C03638=1065.158,313.293,401.347,173.947,33.225,156.127
C03639=1065.152,313.045,401.379,173.944,33.220,156.126
C03640=1065.146,312.797,401.412,173.941,33.216,156.125
C03641=1065.139,312.550,401.445,173.938,33.212,156.124
C03642=1065.133,312.302,401.478,173.934,33.207,156.124
C03643=1065.126,312.054,401.509,173.931,33.203,156.123
C03644=1065.120,311.806,401.542,173.928,33.199,156.122
C03645=1065.113,311.558,401.575,173.925,33.195,156.121
C03646=1065.107,311.311,401.608,173.922,33.190,156.120
C03647=1065.101,311.063,401.640,173.919,33.186,156.119
C03648=1065.094,310.816,401.673,173.915,33.181,156.118
C03649=1065.088,310.568,401.706,173.912,33.177,156.118
C03650=1065.082,310.320,401.738,173.909,33.173,156.117
C03651=1065.076,310.072,401.771,173.906,33.169,156.116
C03652=1065.069,309.824,401.804,173.903,33.165,156.115
C03653=1065.062,309.577,401.836,173.900,33.160,156.114
C03654=1065.056,309.328,401.868,173.897,33.156,156.113
C03655=1065.050,309.081,401.901,173.894,33.151,156.113
C03656=1065.043,308.833,401.933,173.890,33.147,156.112
C03657=1065.037,308.585,401.966,173.887,33.143,156.111
C03658=1065.031,308.337,401.998,173.884,33.139,156.110
C03659=1065.025,308.090,402.031,173.881,33.134,156.109
C03660=1065.019,307.842,402.063,173.877,33.130,156.108
C03661=1065.012,307.594,402.095,173.874,33.126,156.108
C03662=1065.005,307.347,402.128,173.871,33.121,156.107
C03663=1064.999,307.099,402.160,173.868,33.117,156.106
C03664=1064.993,306.851,402.193,173.865,33.113,156.105
C03665=1064.987,306.603,402.225,173.862,33.109,156.104
C03666=1064.981,306.355,402.257,173.859,33.104,156.103
C03667=1064.974,306.108,402.290,173.855,33.100,156.103
C03668=1064.968,305.860,402.322,173.852,33.095,156.102
C03669=1064.962,305.613,402.354,173.849,33.091,156.101
C03670=1064.956,305.365,402.386,173.846,33.087,156.100
C03671=1064.950,305.117,402.419,173.843,33.083,156.099
C03672=1064.943,304.882,402.449,173.840,33.079,156.099
C03673=1064.938,304.648,402.479,173.837,33.074,156.098
C03674=1064.932,304.413,402.510,173.835,33.071,156.097
C03675=1064.927,304.179,402.540,173.832,33.067,156.096
C03676=1064.920,303.944,402.571,173.829,33.062,156.095
C03677=1064.914,303.710,402.600,173.826,33.058,156.095
C03678=1064.908,303.476,402.631,173.823,33.055,156.094
C03679=1064.903,303.241,402.661,173.820,33.050,156.093
C03680=1064.897,302.994,402.694,173.817,33.046,156.092
C03681=1064.890,302.746,402.726,173.814,33.042,156.091
C03682=1064.884,302.498,402.758,173.811,33.038,156.091
C03683=1064.878,302.250,402.790,173.808,33.033,156.090
C03684=1064.872,302.002,402.822,173.805,33.029,156.089
C03685=1064.866,301.755,402.853,173.802,33.025,156.088
C03686=1064.860,301.506,402.885,173.799,33.021,156.087
C03687=1064.853,301.259,402.918,173.796,33.016,156.086
C03688=1064.847,301.011,402.950,173.793,33.012,156.086
C03689=1064.841,300.763,402.981,173.790,33.008,156.085
C03690=1064.835,300.515,403.013,173.787,33.003,156.084
C03691=1064.829,300.268,403.046,173.784,32.999,156.083
C03692=1064.824,300.020,403.078,173.781,32.995,156.082
C03693=1064.817,299.772,403.109,173.778,32.991,156.082
C03694=1064.811,299.524,403.141,173.775,32.986,156.081
C03695=1064.805,299.276,403.173,173.772,32.982,156.080
C03696=1064.800,299.028,403.205,173.769,32.978,156.079
C03697=1064.793,298.780,403.236,173.766,32.974,156.078
C03698=1064.787,298.532,403.268,173.763,32.970,156.077
C03699=1064.781,298.285,403.300,173.760,32.965,156.077
C03700=1064.775,298.037,403.331,173.757,32.961,156.076
C03701=1064.769,297.788,403.363,173.754,32.957,156.075
C03702=1064.763,297.541,403.395,173.751,32.953,156.074
C03703=1064.756,297.294,403.427,173.748,32.948,156.073
C03704=1064.751,297.045,403.459,173.745,32.944,156.073
C03705=1064.745,296.798,403.490,173.742,32.940,156.072
C03706=1064.739,296.549,403.522,173.739,32.936,156.071
C03707=1064.732,296.301,403.553,173.737,32.932,156.070
C03708=1064.726,296.053,403.585,173.734,32.927,156.069
C03709=1064.720,295.806,403.616,173.731,32.923,156.069
C03710=1064.714,295.558,403.648,173.728,32.919,156.068
C03711=1064.707,295.310,403.680,173.725,32.915,156.067
C03712=1064.702,295.062,403.711,173.722,32.911,156.066
C03713=1064.695,294.814,403.742,173.719,32.907,156.065
C03714=1064.688,294.566,403.773,173.716,32.902,156.065
C03715=1064.683,294.319,403.805,173.713,32.898,156.064
C03716=1064.676,294.071,403.837,173.710,32.894,156.063
C03717=1064.670,293.822,403.867,173.707,32.890,156.062
C03718=1064.664,293.575,403.898,173.704,32.886,156.061
C03719=1064.658,293.327,403.930,173.701,32.882,156.061
C03720=1064.651,293.078,403.961,173.698,32.878,156.060
C03721=1064.645,292.831,403.992,173.695,32.873,156.059
C03722=1064.639,292.583,404.024,173.692,32.870,156.058
C03723=1064.633,292.335,404.055,173.690,32.865,156.058
C03724=1064.625,292.001,404.096,173.686,32.860,156.056
C03725=1064.617,291.668,404.139,173.682,32.855,156.055
C03726=1064.609,291.334,404.181,173.678,32.848,156.054
C03727=1064.600,291.000,404.223,173.674,32.843,156.053
C03728=1064.591,290.631,404.269,173.670,32.837,156.052
C03729=1064.582,290.264,404.316,173.665,32.831,156.051
C03730=1064.572,289.896,404.361,173.661,32.825,156.050
C03731=1064.563,289.528,404.407,173.657,32.819,156.049
C03732=1064.557,289.280,404.438,173.654,32.815,156.048
C03733=1064.551,289.032,404.468,173.651,32.811,156.047
C03734=1064.545,288.784,404.500,173.648,32.807,156.046
C03735=1064.539,288.536,404.531,173.645,32.802,156.046
C03736=1064.532,288.288,404.562,173.642,32.799,156.045
C03737=1064.527,288.040,404.593,173.639,32.794,156.044
C03738=1064.520,287.792,404.623,173.637,32.790,156.043
C03739=1064.514,287.545,404.654,173.634,32.786,156.043
C03740=1064.508,287.296,404.685,173.631,32.782,156.042
C03741=1064.502,287.048,404.715,173.628,32.778,156.041
C03742=1064.495,286.800,404.747,173.625,32.774,156.040
C03743=1064.489,286.553,404.777,173.622,32.770,156.039
C03744=1064.483,286.304,404.808,173.620,32.766,156.039
C03745=1064.477,286.056,404.838,173.618,32.762,156.038
C03746=1064.470,285.808,404.870,173.615,32.758,156.037
C03747=1064.464,285.560,404.900,173.612,32.754,156.036
C03748=1064.458,285.312,404.931,173.609,32.750,156.036
C03749=1064.452,285.064,404.961,173.606,32.746,156.035
C03750=1064.446,284.816,404.992,173.603,32.742,156.034
C03751=1064.440,284.568,405.023,173.601,32.738,156.033
C03752=1064.434,284.321,405.053,173.598,32.734,156.033
C03753=1064.427,284.072,405.084,173.595,32.730,156.032
C03754=1064.422,283.824,405.114,173.592,32.726,156.031
C03755=1064.415,283.576,405.145,173.589,32.722,156.030
C03756=1064.409,283.328,405.175,173.586,32.718,156.030
C03757=1064.404,283.080,405.206,173.584,32.713,156.029
C03758=1064.397,282.832,405.236,173.581,32.710,156.028
C03759=1064.391,282.584,405.267,173.578,32.705,156.027
C03760=1064.385,282.335,405.298,173.575,32.701,156.026
C03761=1064.379,282.087,405.328,173.572,32.697,156.026
C03762=1064.373,281.840,405.358,173.570,32.693,156.025
C03763=1064.366,281.591,405.388,173.567,32.689,156.024
C03764=1064.360,281.344,405.419,173.564,32.685,156.023
C03765=1064.355,281.096,405.449,173.561,32.681,156.023
C03766=1064.348,280.847,405.480,173.558,32.677,156.022
C03767=1064.342,280.599,405.510,173.556,32.673,156.021
C03768=1064.336,280.352,405.540,173.553,32.669,156.020
C03769=1064.330,280.103,405.571,173.550,32.665,156.020
C03770=1064.324,279.855,405.602,173.547,32.661,156.019
C03771=1064.318,279.608,405.631,173.545,32.657,156.018
C03772=1064.311,279.359,405.662,173.543,32.653,156.017
C03773=1064.306,279.111,405.692,173.540,32.649,156.017
C03774=1064.300,278.863,405.722,173.537,32.645,156.016
C03775=1064.293,278.615,405.752,173.534,32.641,156.015
C03776=1064.287,278.367,405.782,173.532,32.637,156.014
C03777=1064.281,278.119,405.813,173.529,32.633,156.014
C03778=1064.274,277.870,405.842,173.526,32.629,156.013
C03779=1064.268,277.622,405.873,173.523,32.625,156.012
C03780=1064.263,277.401,405.900,173.521,32.621,156.011
C03781=1064.257,277.179,405.927,173.518,32.618,156.011
C03782=1064.252,276.958,405.953,173.516,32.614,156.010
C03783=1064.247,276.736,405.980,173.514,32.611,156.009
C03784=1064.242,276.514,406.007,173.511,32.607,156.009
C03785=1064.236,276.293,406.034,173.509,32.603,156.008
C03786=1064.230,276.071,406.060,173.506,32.600,156.007
C03787=1064.224,275.850,406.088,173.504,32.597,156.007
C03788=1064.219,275.601,406.117,173.501,32.592,156.006
C03789=1064.213,275.353,406.148,173.498,32.589,156.005
C03790=1064.207,275.105,406.177,173.496,32.585,156.005
C03791=1064.200,274.857,406.207,173.493,32.581,156.004
C03792=1064.194,274.609,406.237,173.490,32.577,156.003
C03793=1064.188,274.361,406.267,173.488,32.573,156.002
C03794=1064.182,274.113,406.297,173.486,32.569,156.002
C03795=1064.176,273.865,406.326,173.483,32.565,156.001
C03796=1064.170,273.616,406.357,173.480,32.561,156.000
C03797=1064.164,273.368,406.386,173.477,32.556,155.999
C03798=1064.158,273.120,406.416,173.475,32.553,155.999
C03799=1064.152,272.872,406.446,173.472,32.548,155.998
C03800=1064.146,272.624,406.476,173.469,32.545,155.997
C03801=1064.140,272.375,406.506,173.467,32.541,155.996
C03802=1064.133,272.128,406.535,173.464,32.537,155.996
C03803=1064.127,271.880,406.564,173.461,32.533,155.995
C03804=1064.121,271.631,406.594,173.459,32.529,155.994
C03805=1064.115,271.384,406.624,173.456,32.525,155.993
C03806=1064.109,271.135,406.653,173.453,32.521,155.993
C03807=1064.102,270.886,406.683,173.450,32.517,155.992
C03808=1064.097,270.639,406.713,173.448,32.513,155.991
C03809=1064.090,270.390,406.742,173.445,32.509,155.991
C03810=1064.085,270.142,406.772,173.443,32.505,155.990
C03811=1064.078,269.894,406.802,173.441,32.501,155.989
C03812=1064.072,269.646,406.831,173.438,32.497,155.988
C03813=1064.066,269.398,406.860,173.435,32.493,155.988
C03814=1064.060,269.150,406.889,173.433,32.490,155.987
C03815=1064.054,268.901,406.920,173.430,32.485,155.986
C03816=1064.048,268.653,406.949,173.427,32.481,155.985
C03817=1064.041,268.405,406.978,173.425,32.477,155.985
C03818=1064.036,268.157,407.008,173.422,32.474,155.984
C03819=1064.030,267.908,407.037,173.419,32.469,155.983
C03820=1064.023,267.661,407.067,173.417,32.466,155.982
C03821=1064.017,267.412,407.096,173.414,32.462,155.982
C03822=1064.011,267.164,407.125,173.411,32.458,155.981
C03823=1064.005,266.916,407.154,173.409,32.454,155.980
C03824=1063.999,266.668,407.183,173.406,32.450,155.979
C03825=1063.993,266.420,407.213,173.404,32.446,155.979
C03826=1063.987,266.171,407.242,173.402,32.442,155.978
C03827=1063.980,265.923,407.271,173.399,32.438,155.977
C03828=1063.975,265.674,407.301,173.396,32.434,155.977
C03829=1063.968,265.426,407.330,173.394,32.430,155.976
C03830=1063.962,265.178,407.359,173.391,32.426,155.975
C03831=1063.956,264.930,407.388,173.389,32.422,155.974
C03832=1063.950,264.681,407.418,173.386,32.418,155.974
C03833=1063.944,264.433,407.447,173.383,32.414,155.973
C03834=1063.938,264.185,407.476,173.381,32.410,155.972
C03835=1063.932,263.937,407.505,173.378,32.406,155.971
C03836=1063.926,263.718,407.531,173.376,32.403,155.971
C03837=1063.921,263.498,407.557,173.373,32.399,155.970
C03838=1063.916,263.278,407.583,173.371,32.396,155.969
C03839=1063.910,263.058,407.608,173.370,32.393,155.969
C03840=1063.905,262.838,407.634,173.367,32.389,155.968
C03841=1063.899,262.619,407.659,173.365,32.386,155.968
C03842=1063.894,262.398,407.685,173.363,32.382,155.967
C03843=1063.888,262.179,407.710,173.360,32.379,155.966
C03844=1063.882,261.930,407.739,173.358,32.375,155.966
C03845=1063.875,261.682,407.768,173.355,32.371,155.965
C03846=1063.869,261.434,407.797,173.353,32.367,155.964
C03847=1063.863,261.185,407.826,173.350,32.364,155.964
C03848=1063.857,260.937,407.855,173.347,32.359,155.963
C03849=1063.851,260.689,407.884,173.345,32.356,155.962
C03850=1063.844,260.441,407.913,173.342,32.352,155.961
C03851=1063.838,260.192,407.941,173.340,32.348,155.961
C03852=1063.832,259.944,407.970,173.338,32.344,155.960
C03853=1063.826,259.696,407.999,173.335,32.340,155.959
C03854=1063.819,259.448,408.028,173.333,32.336,155.958
C03855=1063.813,259.199,408.056,173.330,32.332,155.958
C03856=1063.807,258.951,408.085,173.328,32.328,155.957
C03857=1063.801,258.703,408.113,173.325,32.324,155.956
C03858=1063.795,258.455,408.142,173.322,32.320,155.956
C03859=1063.789,258.207,408.171,173.320,32.317,155.955
C03860=1063.783,257.958,408.199,173.317,32.313,155.954
C03861=1063.777,257.710,408.228,173.315,32.309,155.953
C03862=1063.771,257.461,408.257,173.312,32.305,155.953
C03863=1063.764,257.214,408.285,173.310,32.301,155.952
C03864=1063.758,256.965,408.314,173.308,32.297,155.951
C03865=1063.752,256.717,408.343,173.305,32.293,155.951
C03866=1063.745,256.469,408.372,173.303,32.289,155.950
C03867=1063.740,256.221,408.400,173.300,32.285,155.949
C03868=1063.734,255.972,408.429,173.298,32.282,155.948
C03869=1063.728,255.724,408.457,173.295,32.277,155.948
C03870=1063.721,255.476,408.485,173.293,32.274,155.947
C03871=1063.715,255.227,408.514,173.290,32.270,155.946
C03872=1063.709,254.979,408.543,173.288,32.266,155.946
C03873=1063.703,254.730,408.571,173.285,32.262,155.945
C03874=1063.697,254.482,408.599,173.283,32.258,155.944
C03875=1063.691,254.234,408.628,173.281,32.254,155.943
C03876=1063.685,253.985,408.656,173.278,32.250,155.943
C03877=1063.678,253.737,408.685,173.276,32.246,155.942
C03878=1063.672,253.489,408.713,173.273,32.242,155.941
C03879=1063.667,253.241,408.741,173.271,32.238,155.941
C03880=1063.661,252.992,408.770,173.268,32.234,155.940
C03881=1063.655,252.744,408.798,173.266,32.231,155.939
C03882=1063.648,252.495,408.826,173.263,32.226,155.938
C03883=1063.642,252.248,408.855,173.261,32.223,155.938
C03884=1063.636,251.999,408.883,173.259,32.219,155.937
C03885=1063.630,251.750,408.911,173.257,32.215,155.936
C03886=1063.625,251.502,408.940,173.254,32.211,155.935
C03887=1063.619,251.254,408.968,173.252,32.207,155.935
C03888=1063.612,251.006,408.996,173.249,32.203,155.934
C03889=1063.606,250.757,409.025,173.247,32.199,155.933
C03890=1063.601,250.509,409.053,173.244,32.195,155.933
C03891=1063.595,250.261,409.082,173.242,32.191,155.932
C03892=1063.589,250.040,409.106,173.240,32.187,155.931
C03893=1063.584,249.819,409.131,173.237,32.184,155.931
C03894=1063.578,249.598,409.157,173.236,32.181,155.930
C03895=1063.574,249.378,409.182,173.234,32.177,155.929
C03896=1063.568,249.157,409.207,173.232,32.173,155.929
C03897=1063.563,248.935,409.231,173.230,32.170,155.928
C03898=1063.558,248.714,409.256,173.227,32.166,155.927
C03899=1063.552,248.493,409.282,173.225,32.163,155.927
C03900=1063.546,248.245,409.309,173.223,32.158,155.926
C03901=1063.540,247.997,409.338,173.220,32.155,155.925
C03902=1063.534,247.748,409.367,173.218,32.150,155.924
C03903=1063.529,247.500,409.394,173.215,32.147,155.924
C03904=1063.522,247.252,409.422,173.214,32.142,155.923
C03905=1063.517,247.004,409.450,173.211,32.139,155.922
C03906=1063.511,246.755,409.478,173.209,32.135,155.922
C03907=1063.505,246.506,409.507,173.206,32.131,155.921
C03908=1063.499,246.259,409.534,173.204,32.127,155.920
C03909=1063.493,246.010,409.562,173.202,32.123,155.919
C03910=1063.486,245.761,409.590,173.199,32.119,155.919
C03911=1063.481,245.513,409.618,173.197,32.115,155.918
C03912=1063.474,245.265,409.646,173.194,32.111,155.917
C03913=1063.469,245.017,409.674,173.193,32.107,155.916
C03914=1063.462,244.768,409.701,173.190,32.103,155.916
C03915=1063.456,244.519,409.729,173.188,32.099,155.915
C03916=1063.450,244.271,409.757,173.185,32.095,155.914
C03917=1063.444,244.023,409.785,173.183,32.091,155.914
C03918=1063.438,243.775,409.812,173.181,32.088,155.913
C03919=1063.432,243.526,409.841,173.178,32.083,155.912
C03920=1063.426,243.278,409.868,173.176,32.080,155.911
C03921=1063.421,243.029,409.896,173.174,32.076,155.911
C03922=1063.414,242.781,409.923,173.172,32.072,155.910
C03923=1063.409,242.532,409.951,173.169,32.068,155.909
C03924=1063.402,242.284,409.979,173.167,32.063,155.908
C03925=1063.397,242.036,410.007,173.165,32.060,155.908
C03926=1063.390,241.787,410.034,173.162,32.056,155.907
C03927=1063.384,241.538,410.062,173.160,32.052,155.906
C03928=1063.378,241.290,410.090,173.157,32.048,155.906
C03929=1063.372,241.041,410.117,173.155,32.044,155.905
C03930=1063.366,240.794,410.144,173.154,32.040,155.904
C03931=1063.359,240.545,410.172,173.151,32.036,155.904
C03932=1063.354,240.297,410.199,173.149,32.033,155.903
C03933=1063.347,240.048,410.227,173.146,32.028,155.902
C03934=1063.341,239.800,410.254,173.144,32.025,155.901
C03935=1063.336,239.551,410.282,173.141,32.021,155.901
C03936=1063.329,239.303,410.309,173.139,32.017,155.900
C03937=1063.323,239.054,410.336,173.137,32.013,155.899
C03938=1063.317,238.806,410.364,173.135,32.008,155.898
C03939=1063.311,238.558,410.392,173.133,32.005,155.898
C03940=1063.305,238.309,410.419,173.131,32.001,155.897
C03941=1063.299,238.061,410.446,173.128,31.997,155.896
C03942=1063.292,237.812,410.473,173.126,31.993,155.896
C03943=1063.286,237.564,410.501,173.123,31.989,155.895
C03944=1063.281,237.315,410.528,173.121,31.985,155.894
C03945=1063.275,237.067,410.555,173.120,31.981,155.893
C03946=1063.268,236.818,410.583,173.117,31.978,155.893
C03947=1063.262,236.570,410.610,173.115,31.973,155.892
C03948=1063.257,236.345,410.634,173.113,31.970,155.891
C03949=1063.251,236.121,410.659,173.111,31.966,155.891
C03950=1063.246,235.898,410.684,173.108,31.963,155.890
C03951=1063.241,235.673,410.708,173.106,31.959,155.889
C03952=1063.235,235.449,410.733,173.104,31.955,155.889
C03953=1063.230,235.226,410.757,173.103,31.952,155.888
C03954=1063.224,235.002,410.781,173.101,31.949,155.888
C03955=1063.219,234.777,410.806,173.099,31.945,155.887
C03956=1063.213,234.529,410.833,173.096,31.940,155.886
C03957=1063.206,234.281,410.861,173.094,31.937,155.885
C03958=1063.201,234.032,410.887,173.092,31.933,155.885
C03959=1063.195,233.784,410.914,173.089,31.929,155.884
C03960=1063.189,233.535,410.942,173.087,31.925,155.883
C03961=1063.183,233.287,410.969,173.086,31.921,155.882
C03962=1063.177,233.038,410.996,173.083,31.917,155.882
C03963=1063.171,232.790,411.023,173.081,31.913,155.881
C03964=1063.165,232.542,411.050,173.079,31.909,155.880
C03965=1063.159,232.293,411.077,173.076,31.905,155.880
C03966=1063.153,232.044,411.104,173.074,31.901,155.879
C03967=1063.147,231.796,411.131,173.072,31.897,155.878
C03968=1063.140,231.547,411.158,173.070,31.893,155.877
C03969=1063.135,231.299,411.185,173.068,31.889,155.877
C03970=1063.129,231.051,411.211,173.066,31.886,155.876
C03971=1063.122,230.802,411.238,173.063,31.881,155.875
C03972=1063.116,230.554,411.266,173.061,31.877,155.875
C03973=1063.111,230.305,411.292,173.059,31.873,155.874
C03974=1063.104,230.056,411.319,173.056,31.869,155.873
C03975=1063.098,229.808,411.346,173.055,31.865,155.872
C03976=1063.093,229.560,411.373,173.053,31.861,155.872
C03977=1063.086,229.311,411.400,173.051,31.858,155.871
C03978=1063.080,229.062,411.426,173.048,31.853,155.870
C03979=1063.074,228.813,411.453,173.046,31.850,155.870
C03980=1063.068,228.565,411.480,173.044,31.845,155.869
C03981=1063.062,228.317,411.506,173.042,31.842,155.868
C03982=1063.055,228.068,411.533,173.040,31.838,155.867
C03983=1063.050,227.819,411.560,173.038,31.834,155.867
C03984=1063.044,227.571,411.586,173.035,31.830,155.866
C03985=1063.038,227.322,411.613,173.033,31.826,155.865
C03986=1063.031,227.074,411.640,173.031,31.822,155.864
C03987=1063.025,226.826,411.666,173.029,31.818,155.864
C03988=1063.019,226.577,411.693,173.027,31.814,155.863
C03989=1063.013,226.328,411.720,173.025,31.810,155.862
C03990=1063.007,226.080,411.747,173.023,31.806,155.862
C03991=1063.001,225.832,411.773,173.020,31.802,155.861
C03992=1062.994,225.583,411.800,173.018,31.798,155.860
C03993=1062.989,225.334,411.826,173.016,31.794,155.859
C03994=1062.983,225.086,411.853,173.014,31.790,155.859
C03995=1062.976,224.838,411.879,173.012,31.786,155.858
C03996=1062.970,224.589,411.906,173.010,31.782,155.857
C03997=1062.964,224.340,411.933,173.008,31.778,155.857
C03998=1062.959,224.091,411.959,173.005,31.774,155.856
C03999=1062.953,223.843,411.985,173.003,31.770,155.855
C04000=1062.946,223.595,412.011,173.001,31.766,155.854
C04001=1062.940,223.346,412.038,173.000,31.762,155.854
C04002=1062.934,223.098,412.065,172.997,31.758,155.853
C04003=1062.929,222.849,412.091,172.995,31.754,155.852
C04004=1062.923,222.621,412.115,172.993,31.751,155.852
C04005=1062.917,222.393,412.139,172.991,31.747,155.851
C04006=1062.913,222.165,412.163,172.989,31.743,155.850
C04007=1062.906,221.937,412.188,172.988,31.740,155.850
C04008=1062.901,221.709,412.212,172.986,31.736,155.849
C04009=1062.896,221.481,412.236,172.984,31.732,155.848
C04010=1062.890,221.253,412.260,172.982,31.728,155.848
C04011=1062.884,221.025,412.285,172.980,31.725,155.847
C04012=1062.878,220.777,412.311,172.978,31.720,155.846
C04013=1062.872,220.528,412.337,172.976,31.717,155.845
C04014=1062.866,220.279,412.363,172.974,31.713,155.845
C04015=1062.860,220.031,412.389,172.972,31.709,155.844
C04016=1062.854,219.782,412.415,172.970,31.705,155.843
C04017=1062.847,219.534,412.442,172.967,31.701,155.843
C04018=1062.842,219.285,412.468,172.965,31.697,155.842
C04019=1062.835,219.037,412.494,172.964,31.693,155.841
C04020=1062.830,218.788,412.520,172.962,31.689,155.840
C04021=1062.823,218.540,412.546,172.959,31.684,155.840
C04022=1062.817,218.291,412.572,172.957,31.681,155.839
C04023=1062.811,218.043,412.598,172.955,31.677,155.838
C04024=1062.805,217.794,412.625,172.953,31.673,155.837
C04025=1062.799,217.545,412.650,172.952,31.669,155.837
C04026=1062.793,217.297,412.677,172.949,31.665,155.836
C04027=1062.787,217.048,412.702,172.947,31.661,155.835
C04028=1062.781,216.800,412.729,172.945,31.657,155.835
C04029=1062.775,216.551,412.754,172.943,31.653,155.834
C04030=1062.769,216.302,412.781,172.941,31.649,155.833
C04031=1062.763,216.054,412.806,172.939,31.645,155.832
C04032=1062.757,215.805,412.833,172.937,31.640,155.832
C04033=1062.751,215.557,412.858,172.935,31.637,155.831
C04034=1062.745,215.308,412.883,172.933,31.632,155.830
C04035=1062.738,215.059,412.910,172.931,31.628,155.829
C04036=1062.732,214.810,412.936,172.929,31.624,155.829
C04037=1062.726,214.562,412.962,172.927,31.620,155.828
C04038=1062.720,214.313,412.988,172.925,31.616,155.827
C04039=1062.714,214.064,413.014,172.923,31.612,155.827
C04040=1062.708,213.816,413.040,172.921,31.608,155.826
C04041=1062.703,213.567,413.065,172.919,31.604,155.825
C04042=1062.696,213.319,413.091,172.917,31.600,155.824
C04043=1062.690,213.071,413.117,172.915,31.596,155.824
C04044=1062.684,212.822,413.143,172.913,31.592,155.823
C04045=1062.678,212.573,413.168,172.911,31.588,155.822
C04046=1062.672,212.325,413.195,172.909,31.584,155.821
C04047=1062.666,212.076,413.220,172.907,31.580,155.821
C04048=1062.660,211.827,413.245,172.905,31.576,155.820
C04049=1062.654,211.579,413.271,172.903,31.572,155.819
C04050=1062.648,211.330,413.297,172.901,31.568,155.818
C04051=1062.642,211.082,413.323,172.899,31.564,155.818
C04052=1062.636,210.833,413.348,172.897,31.560,155.817
C04053=1062.630,210.584,413.374,172.896,31.555,155.816
C04054=1062.624,210.335,413.399,172.893,31.551,155.816
C04055=1062.618,210.087,413.425,172.891,31.547,155.815
C04056=1062.611,209.839,413.451,172.889,31.543,155.814
C04057=1062.606,209.590,413.477,172.887,31.539,155.813
C04058=1062.599,209.341,413.502,172.886,31.535,155.813
C04059=1062.594,209.093,413.527,172.884,31.531,155.812
C04060=1062.588,208.867,413.551,172.882,31.527,155.811
C04061=1062.583,208.641,413.573,172.880,31.524,155.811
C04062=1062.578,208.416,413.597,172.878,31.520,155.810
C04063=1062.572,208.190,413.620,172.877,31.516,155.809
C04064=1062.566,207.965,413.643,172.875,31.512,155.808
C04065=1062.561,207.740,413.665,172.873,31.509,155.808
C04066=1062.555,207.514,413.689,172.871,31.505,155.807
C04067=1062.550,207.288,413.712,172.869,31.501,155.806
C04068=1062.524,206.240,413.816,172.699,31.419,155.799
C04069=1062.519,205.992,413.840,172.697,31.416,155.799
C04070=1062.513,205.742,413.865,172.694,31.413,155.798
C04071=1062.507,205.494,413.890,172.692,31.410,155.797
C04072=1062.502,205.245,413.914,172.690,31.407,155.797
C04073=1062.496,204.997,413.939,172.688,31.403,155.796
C04074=1062.489,204.748,413.963,172.686,31.400,155.796
C04075=1062.484,204.500,413.988,172.683,31.397,155.795
C04076=1062.478,204.250,414.012,172.681,31.394,155.795
C04077=1062.473,204.002,414.036,172.678,31.390,155.794
C04078=1062.467,203.753,414.062,172.676,31.387,155.794
C04079=1062.461,203.504,414.086,172.675,31.384,155.793
C04080=1062.455,203.255,414.110,172.672,31.381,155.793
C04081=1062.449,203.007,414.134,172.670,31.378,155.792
C04082=1062.443,202.758,414.159,172.667,31.375,155.792
C04083=1062.438,202.510,414.184,172.665,31.372,155.791
C04084=1062.432,202.260,414.209,172.663,31.369,155.791
C04085=1062.426,202.012,414.232,172.661,31.365,155.790
C04086=1062.420,201.763,414.257,172.659,31.362,155.790
C04087=1062.415,201.514,414.281,172.656,31.359,155.789
C04088=1062.408,201.265,414.305,172.654,31.356,155.789
C04089=1062.403,201.017,414.329,172.651,31.353,155.788
C04090=1062.396,200.768,414.353,172.650,31.350,155.787
C04091=1062.391,200.519,414.378,172.648,31.347,155.787
C04092=1062.384,200.270,414.402,172.645,31.344,155.787
C04093=1062.379,200.021,414.426,172.643,31.340,155.786
C04094=1062.372,199.773,414.450,172.640,31.337,155.785
C04095=1062.367,199.524,414.474,172.638,31.335,155.785
C04096=1062.361,199.276,414.498,172.637,31.331,155.784
C04097=1062.355,199.026,414.522,172.634,31.328,155.784
C04098=1062.349,198.778,414.546,172.632,31.325,155.784
C04099=1062.343,198.529,414.571,172.629,31.322,155.783
C04100=1062.337,198.281,414.594,172.627,31.319,155.782
C04101=1062.331,198.031,414.619,172.626,31.316,155.782
C04102=1062.325,197.783,414.643,172.623,31.313,155.782
C04103=1062.319,197.534,414.667,172.621,31.310,155.781
C04104=1062.313,197.285,414.691,172.619,31.307,155.780
C04105=1062.308,197.037,414.715,172.616,31.304,155.780
C04106=1062.301,196.788,414.739,172.614,31.301,155.780
C04107=1062.296,196.539,414.764,172.612,31.297,155.779
C04108=1062.290,196.291,414.787,172.610,31.295,155.779
C04109=1062.284,196.042,414.812,172.608,31.292,155.778
C04110=1062.278,195.793,414.835,172.605,31.288,155.777
C04111=1062.272,195.543,414.859,172.603,31.286,155.777
C04112=1062.266,195.295,414.883,172.602,31.282,155.777
C04113=1062.261,195.047,414.907,172.599,31.279,155.776
C04114=1062.254,194.798,414.931,172.597,31.276,155.776
C04115=1062.249,194.548,414.955,172.595,31.273,155.775
C04116=1062.243,194.300,414.979,172.592,31.270,155.775
C04117=1062.237,194.051,415.003,172.591,31.267,155.774
C04118=1062.231,193.803,415.027,172.589,31.264,155.774
C04119=1062.226,193.554,415.051,172.586,31.261,155.773
C04120=1062.220,193.304,415.074,172.584,31.258,155.772
C04121=1062.215,193.056,415.099,172.582,31.255,155.772
C04122=1062.208,192.808,415.122,172.579,31.252,155.772
C04123=1062.203,192.559,415.145,172.578,31.248,155.771
C04124=1062.197,192.309,415.170,172.576,31.246,155.771
C04125=1062.191,192.061,415.194,172.573,31.242,155.770
C04126=1062.186,191.812,415.217,172.571,31.239,155.770
C04127=1062.180,191.564,415.241,172.569,31.237,155.769
C04128=1062.174,191.314,415.265,172.567,31.233,155.769
C04129=1062.167,191.031,415.291,172.565,31.230,155.768
C04130=1062.161,190.748,415.319,172.562,31.226,155.767
C04131=1062.154,190.465,415.346,172.560,31.223,155.767
C04132=1062.147,190.181,415.373,172.557,31.220,155.766
C04133=1062.142,189.932,415.397,172.556,31.216,155.766
C04134=1062.136,189.684,415.420,172.553,31.213,155.765
C04135=1062.131,189.435,415.444,172.551,31.211,155.765
C04136=1062.125,189.187,415.468,172.549,31.207,155.764
C04137=1062.118,188.937,415.491,172.546,31.205,155.764
C04138=1062.113,188.689,415.515,172.545,31.201,155.763
C04139=1062.107,188.440,415.538,172.543,31.198,155.763
C04140=1062.101,188.191,415.562,172.541,31.196,155.762
C04141=1062.096,187.942,415.586,172.538,31.192,155.762
C04142=1062.090,187.694,415.609,172.536,31.189,155.761
C04143=1062.085,187.444,415.633,172.535,31.186,155.761
C04144=1062.079,187.196,415.657,172.533,31.183,155.760
C04145=1062.073,186.947,415.680,172.530,31.180,155.760
C04146=1062.068,186.698,415.704,172.528,31.177,155.759
C04147=1062.062,186.449,415.727,172.526,31.174,155.759
C04148=1062.057,186.201,415.751,172.524,31.171,155.758
C04149=1062.051,185.952,415.774,172.522,31.168,155.758
C04150=1062.045,185.703,415.797,172.520,31.165,155.757
C04151=1062.039,185.454,415.822,172.518,31.162,155.757
C04152=1062.034,185.205,415.845,172.515,31.159,155.756
C04153=1062.028,184.956,415.868,172.513,31.156,155.756
C04154=1062.023,184.707,415.892,172.512,31.152,155.755
C04155=1062.017,184.458,415.915,172.510,31.150,155.755
C04156=1062.011,184.210,415.939,172.507,31.147,155.754
C04157=1062.004,183.960,415.962,172.505,31.144,155.754
C04158=1061.999,183.712,415.985,172.503,31.141,155.754
C04159=1061.993,183.463,416.008,172.502,31.138,155.753
C04160=1061.987,183.214,416.031,172.499,31.135,155.753
C04161=1061.980,182.966,416.054,172.497,31.133,155.752
C04162=1061.974,182.716,416.077,172.495,31.129,155.752
C04163=1061.968,182.467,416.100,172.493,31.127,155.751
C04164=1061.962,182.219,416.124,172.491,31.124,155.751
C04165=1061.957,181.970,416.147,172.489,31.121,155.750
C04166=1061.951,181.721,416.170,172.487,31.118,155.750
C04167=1061.945,181.472,416.193,172.485,31.116,155.749
C04168=1061.939,181.223,416.216,172.482,31.112,155.749
C04169=1061.933,180.974,416.239,172.480,31.110,155.749
C04170=1061.926,180.726,416.262,172.479,31.106,155.748
C04171=1061.921,180.477,416.285,172.477,31.104,155.748
C04172=1061.915,180.228,416.308,172.474,31.101,155.747
C04173=1061.909,179.979,416.331,172.472,31.098,155.747
C04174=1061.903,179.730,416.354,172.470,31.095,155.746
C04175=1061.897,179.481,416.377,172.469,31.093,155.746
C04176=1061.891,179.232,416.400,172.466,31.089,155.745
C04177=1061.885,178.984,416.423,172.464,31.087,155.745
C04178=1061.879,178.735,416.446,172.462,31.084,155.744
C04179=1061.873,178.486,416.469,172.460,31.081,155.744
C04180=1061.867,178.237,416.492,172.459,31.078,155.743
C04181=1061.862,177.988,416.515,172.456,31.075,155.743
C04182=1061.856,177.739,416.538,172.454,31.072,155.743
C04183=1061.850,177.490,416.561,172.452,31.069,155.742
C04184=1061.844,177.242,416.583,172.450,31.066,155.742
C04185=1061.838,176.993,416.606,172.448,31.063,155.741
C04186=1061.832,176.743,416.629,172.446,31.061,155.741
C04187=1061.826,176.494,416.652,172.444,31.058,155.740
C04188=1061.820,176.246,416.675,172.442,31.055,155.740
C04189=1061.814,175.997,416.698,172.440,31.052,155.739
C04190=1061.808,175.748,416.720,172.438,31.049,155.739
C04191=1061.802,175.499,416.743,172.436,31.046,155.738
C04192=1061.797,175.250,416.766,172.434,31.044,155.738
C04193=1061.790,174.967,416.792,172.432,31.041,155.737
C04194=1061.783,174.683,416.818,172.429,31.037,155.737
C04195=1061.777,174.399,416.843,172.428,31.034,155.736
C04196=1061.770,174.116,416.869,172.425,31.031,155.736
C04197=1061.764,173.867,416.892,172.423,31.027,155.735
C04198=1061.759,173.618,416.915,172.421,31.025,155.735
C04199=1061.753,173.369,416.938,172.419,31.022,155.735
C04200=1061.747,173.121,416.961,172.417,31.019,155.734
C04201=1061.741,172.871,416.983,172.415,31.016,155.734
C04202=1061.735,172.622,417.006,172.413,31.013,155.733
C04203=1061.730,172.373,417.029,172.411,31.010,155.733
C04204=1061.724,172.124,417.052,172.409,31.008,155.732
C04205=1061.717,171.876,417.074,172.408,31.005,155.732
C04206=1061.712,171.626,417.096,172.405,31.002,155.731
C04207=1061.706,171.377,417.119,172.403,30.999,155.731
C04208=1061.701,171.129,417.142,172.401,30.996,155.730
C04209=1061.694,170.880,417.164,172.399,30.993,155.730
C04210=1061.688,170.631,417.187,172.398,30.990,155.730
C04211=1061.683,170.382,417.210,172.396,30.987,155.729
C04212=1061.678,170.133,417.232,172.394,30.985,155.729
C04213=1061.671,169.885,417.255,172.391,30.982,155.728
C04214=1061.666,169.636,417.277,172.389,30.979,155.728
C04215=1061.660,169.386,417.300,172.388,30.976,155.727
C04216=1061.654,169.137,417.323,172.386,30.973,155.727
C04217=1061.648,168.889,417.345,172.384,30.970,155.726
C04218=1061.643,168.639,417.367,172.382,30.967,155.726
C04219=1061.637,168.390,417.390,172.380,30.965,155.725
C04220=1061.632,168.142,417.413,172.379,30.962,155.725
C04221=1061.626,167.893,417.434,172.376,30.959,155.724
C04222=1061.620,167.644,417.457,172.374,30.956,155.724
C04223=1061.614,167.395,417.480,172.372,30.953,155.724
C04224=1061.609,167.146,417.503,172.370,30.950,155.723
C04225=1061.602,166.897,417.525,172.369,30.947,155.723
C04226=1061.597,166.648,417.547,172.367,30.944,155.722
C04227=1061.592,166.399,417.570,172.365,30.942,155.722
C04228=1061.585,166.151,417.592,172.363,30.939,155.721
C04229=1061.580,165.901,417.614,172.360,30.936,155.721
C04230=1061.574,165.652,417.637,172.359,30.933,155.720
C04231=1061.569,165.404,417.659,172.357,30.930,155.720
C04232=1061.563,165.155,417.681,172.355,30.927,155.719
C04233=1061.557,164.906,417.704,172.353,30.924,155.719
C04234=1061.552,164.657,417.727,172.351,30.921,155.718
C04235=1061.546,164.408,417.748,172.350,30.919,155.718
C04236=1061.540,164.159,417.771,172.348,30.916,155.718
C04237=1061.535,163.910,417.793,172.346,30.913,155.717
C04238=1061.528,163.661,417.815,172.344,30.910,155.717
C04239=1061.524,163.412,417.837,172.342,30.907,155.716
C04240=1061.518,163.163,417.860,172.340,30.904,155.716
C04241=1061.512,162.914,417.882,172.338,30.901,155.715
C04242=1061.506,162.665,417.905,172.336,30.898,155.715
C04243=1061.501,162.416,417.927,172.334,30.896,155.714
C04244=1061.495,162.168,417.949,172.333,30.892,155.714
C04245=1061.489,161.918,417.971,172.331,30.890,155.713
C04246=1061.484,161.670,417.993,172.329,30.887,155.713
C04247=1061.478,161.421,418.015,172.327,30.884,155.712
C04248=1061.472,161.171,418.038,172.325,30.881,155.712
C04249=1061.467,160.923,418.061,172.324,30.878,155.712
C04250=1061.461,160.674,418.082,172.322,30.875,155.711
C04251=1061.455,160.425,418.104,172.320,30.873,155.711
C04252=1061.449,160.176,418.126,172.318,30.870,155.710
C04253=1061.443,159.927,418.148,172.315,30.867,155.710
C04254=1061.438,159.678,418.169,172.314,30.864,155.709
C04255=1061.432,159.429,418.192,172.312,30.861,155.709
C04256=1061.426,159.180,418.214,172.310,30.859,155.709
C04257=1061.420,158.896,418.239,172.308,30.856,155.708
C04258=1061.412,158.612,418.264,172.305,30.853,155.708
C04259=1061.406,158.328,418.289,172.304,30.849,155.707
C04260=1061.399,158.044,418.313,172.302,30.846,155.707
C04261=1061.393,157.795,418.336,172.300,30.844,155.706
C04262=1061.387,157.546,418.358,172.298,30.841,155.706
C04263=1061.381,157.297,418.379,172.297,30.838,155.705
C04264=1061.376,157.048,418.401,172.295,30.835,155.705
C04265=1061.370,156.799,418.423,172.292,30.832,155.704
C04266=1061.364,156.550,418.445,172.290,30.830,155.704
C04267=1061.359,156.301,418.467,172.288,30.827,155.704
C04268=1061.353,156.052,418.489,172.287,30.824,155.703
C04269=1061.346,155.803,418.510,172.285,30.821,155.703
C04270=1061.341,155.554,418.531,172.283,30.818,155.702
C04271=1061.335,155.305,418.554,172.281,30.816,155.702
C04272=1061.329,155.056,418.576,172.279,30.813,155.701
C04273=1061.323,154.807,418.598,172.278,30.810,155.701
C04274=1061.317,154.558,418.619,172.276,30.807,155.700
C04275=1061.312,154.309,418.641,172.274,30.805,155.700
C04276=1061.306,154.060,418.663,172.272,30.802,155.700
C04277=1061.300,153.811,418.684,172.270,30.799,155.699
C04278=1061.294,153.562,418.706,172.269,30.797,155.699
C04279=1061.288,153.313,418.727,172.267,30.794,155.698
C04280=1061.282,153.064,418.749,172.265,30.791,155.698
C04281=1061.277,152.815,418.771,172.263,30.788,155.697
C04282=1061.271,152.566,418.792,172.261,30.785,155.697
C04283=1061.265,152.317,418.814,172.260,30.783,155.697
C04284=1061.259,152.068,418.835,172.258,30.780,155.696
C04285=1061.253,151.819,418.857,172.256,30.777,155.696
C04286=1061.247,151.570,418.878,172.254,30.775,155.695
C04287=1061.241,151.321,418.900,172.253,30.772,155.695
C04288=1061.236,151.072,418.922,172.251,30.769,155.694
C04289=1061.230,150.823,418.943,172.249,30.766,155.694
C04290=1061.224,150.574,418.965,172.247,30.764,155.693
C04291=1061.218,150.325,418.986,172.245,30.761,155.693
C04292=1061.212,150.076,419.008,172.244,30.758,155.693
C04293=1061.207,149.827,419.029,172.242,30.756,155.692
C04294=1061.200,149.578,419.051,172.240,30.752,155.692
C04295=1061.195,149.329,419.071,172.238,30.750,155.691
C04296=1061.189,149.080,419.093,172.236,30.747,155.691
C04297=1061.183,148.831,419.115,172.234,30.744,155.690
C04298=1061.177,148.582,419.136,172.232,30.742,155.690
C04299=1061.171,148.333,419.158,172.230,30.739,155.690
C04300=1061.166,148.084,419.179,172.228,30.736,155.689
C04301=1061.160,147.835,419.201,172.227,30.733,155.689
C04302=1061.154,147.585,419.222,172.225,30.730,155.688
C04303=1061.148,147.337,419.243,172.223,30.728,155.688
C04304=1061.142,147.088,419.264,172.221,30.725,155.687
C04305=1061.136,146.839,419.286,172.219,30.722,155.687
C04306=1061.130,146.590,419.307,172.218,30.720,155.687
C04307=1061.125,146.341,419.328,172.216,30.717,155.686
C04308=1061.119,146.092,419.349,172.214,30.714,155.686
C04309=1061.112,145.843,419.371,172.212,30.712,155.685
C04310=1061.107,145.594,419.392,172.211,30.709,155.685
C04311=1061.101,145.344,419.413,172.210,30.707,155.685
C04312=1061.096,145.096,419.435,172.208,30.704,155.684
C04313=1061.089,144.846,419.456,172.206,30.701,155.684
C04314=1061.083,144.598,419.477,172.204,30.699,155.683
C04315=1061.077,144.348,419.498,172.202,30.695,155.683
C04316=1061.072,144.100,419.519,172.201,30.693,155.682
C04317=1061.065,143.851,419.541,172.199,30.690,155.682
C04318=1061.060,143.602,419.561,172.197,30.687,155.682
C04319=1061.054,143.352,419.583,172.195,30.685,155.681
C04320=1061.048,143.104,419.604,172.194,30.682,155.681
C04321=1061.041,142.819,419.628,172.191,30.679,155.680
C04322=1061.035,142.534,419.652,172.189,30.676,155.680
C04323=1061.028,142.250,419.676,172.187,30.673,155.679
C04324=1061.021,141.966,419.700,172.185,30.669,155.679
C04325=1061.015,141.717,419.721,172.184,30.667,155.678
C04326=1061.010,141.468,419.742,172.182,30.664,155.678
C04327=1061.004,141.219,419.764,172.180,30.661,155.677
C04328=1060.998,140.970,419.784,172.178,30.659,155.677
C04329=1060.992,140.721,419.806,172.177,30.656,155.677
C04330=1060.987,140.471,419.826,172.175,30.653,155.676
C04331=1060.980,140.222,419.847,172.173,30.651,155.676
C04332=1060.975,139.974,419.869,172.171,30.648,155.675
C04333=1060.969,139.724,419.890,172.169,30.645,155.675
C04334=1060.963,139.476,419.911,172.168,30.643,155.675
C04335=1060.957,139.227,419.931,172.166,30.640,155.674
C04336=1060.951,138.978,419.952,172.164,30.637,155.674
C04337=1060.946,138.729,419.973,172.162,30.634,155.673
C04338=1060.940,138.479,419.995,172.161,30.631,155.673
C04339=1060.934,138.230,420.015,172.159,30.629,155.672
C04340=1060.928,137.981,420.035,172.157,30.626,155.672
C04341=1060.922,137.732,420.057,172.155,30.623,155.672
C04342=1060.916,137.483,420.077,172.153,30.621,155.671
C04343=1060.910,137.234,420.098,172.153,30.618,155.671
C04344=1060.905,136.985,420.119,172.151,30.616,155.670
C04345=1060.898,136.736,420.140,172.149,30.613,155.670
C04346=1060.893,136.487,420.161,172.147,30.610,155.669
C04347=1060.887,136.237,420.181,172.145,30.608,155.669
C04348=1060.880,135.989,420.202,172.144,30.605,155.669
C04349=1060.875,135.739,420.223,172.142,30.602,155.668
C04350=1060.869,135.490,420.243,172.140,30.600,155.668
C04351=1060.863,135.242,420.264,172.138,30.597,155.667
C04352=1060.857,134.992,420.285,172.137,30.594,155.667
C04353=1060.851,134.743,420.305,172.135,30.592,155.667
C04354=1060.845,134.494,420.327,172.133,30.589,155.666
C04355=1060.840,134.245,420.347,172.131,30.586,155.666
C04356=1060.834,133.996,420.367,172.129,30.584,155.665
C04357=1060.828,133.747,420.389,172.128,30.581,155.665
C04358=1060.822,133.498,420.409,172.127,30.578,155.665
C04359=1060.816,133.249,420.429,172.125,30.576,155.664
C04360=1060.810,133.000,420.451,172.123,30.573,155.664
C04361=1060.804,132.751,420.471,172.122,30.570,155.663
C04362=1060.799,132.502,420.492,172.120,30.568,155.663
C04363=1060.792,132.252,420.512,172.118,30.565,155.662
C04364=1060.787,132.004,420.533,172.116,30.562,155.662
C04365=1060.782,131.755,420.554,172.114,30.559,155.662
C04366=1060.775,131.505,420.574,172.113,30.557,155.661
C04367=1060.769,131.256,420.594,172.111,30.554,155.661
C04368=1060.763,131.006,420.615,172.109,30.552,155.660
C04369=1060.757,130.758,420.636,172.107,30.549,155.660
C04370=1060.751,130.509,420.656,172.106,30.546,155.660
C04371=1060.745,130.260,420.676,172.105,30.544,155.659
C04372=1060.739,130.011,420.696,172.103,30.541,155.659
C04373=1060.732,129.761,420.717,172.101,30.538,155.658
C04374=1060.727,129.512,420.737,172.099,30.536,155.658
C04375=1060.721,129.263,420.757,172.098,30.533,155.657
C04376=1060.715,129.014,420.778,172.096,30.530,155.657
C04377=1060.709,128.765,420.799,172.094,30.528,155.657
C04378=1060.703,128.517,420.819,172.092,30.526,155.656
C04379=1060.696,128.267,420.839,172.091,30.523,155.656
C04380=1060.691,128.018,420.860,172.089,30.520,155.656
C04381=1060.685,127.769,420.880,172.087,30.518,155.655
C04382=1060.679,127.520,420.900,172.086,30.515,155.655
C04383=1060.673,127.270,420.921,172.084,30.512,155.654
C04384=1060.667,127.022,420.940,172.083,30.510,155.654
C04385=1060.660,126.737,420.963,172.081,30.507,155.653
C04386=1060.654,126.453,420.986,172.078,30.504,155.653
C04387=1060.647,126.168,421.010,172.076,30.501,155.653
C04388=1060.640,125.884,421.033,172.075,30.498,155.652
C04389=1060.633,125.635,421.054,172.073,30.495,155.652
C04390=1060.628,125.386,421.074,172.071,30.492,155.651
C04391=1060.622,125.136,421.093,172.069,30.490,155.651
C04392=1060.616,124.887,421.113,172.068,30.487,155.650
C04393=1060.610,124.637,421.134,172.067,30.484,155.650
C04394=1060.604,124.389,421.154,172.065,30.482,155.650
C04395=1060.598,124.140,421.174,172.063,30.479,155.649
C04396=1060.592,123.891,421.194,172.061,30.476,155.649
C04397=1060.587,123.641,421.215,172.060,30.474,155.648
C04398=1060.581,123.392,421.235,172.058,30.472,155.648
C04399=1060.575,123.144,421.255,172.056,30.469,155.648
C04400=1060.569,122.894,421.275,172.054,30.466,155.647
C04401=1060.563,122.645,421.296,172.054,30.464,155.647
C04402=1060.557,122.396,421.316,172.052,30.461,155.646
C04403=1060.551,122.147,421.336,172.050,30.458,155.646
C04404=1060.546,121.898,421.356,172.048,30.456,155.646
C04405=1060.540,121.649,421.375,172.046,30.453,155.645
C04406=1060.533,121.399,421.396,172.045,30.450,155.645
C04407=1060.527,121.150,421.416,172.043,30.448,155.644
C04408=1060.522,120.901,421.436,172.041,30.445,155.644
C04409=1060.516,120.653,421.456,172.040,30.442,155.643
C04410=1060.510,120.403,421.476,172.039,30.440,155.643
C04411=1060.504,120.154,421.496,172.037,30.437,155.643
C04412=1060.498,119.904,421.516,172.035,30.434,155.642
C04413=1060.492,119.656,421.536,172.033,30.432,155.642
C04414=1060.487,119.407,421.556,172.032,30.429,155.641
C04415=1060.481,119.157,421.576,172.030,30.426,155.641
C04416=1060.476,118.908,421.596,172.029,30.424,155.641
C04417=1060.470,118.659,421.616,172.027,30.421,155.640
C04418=1060.463,118.410,421.636,172.025,30.418,155.640
C04419=1060.457,118.160,421.656,172.024,30.416,155.639
C04420=1060.451,117.912,421.676,172.022,30.413,155.639
C04421=1060.446,117.663,421.696,172.020,30.410,155.639
C04422=1060.440,117.414,421.716,172.018,30.408,155.638
C04423=1060.434,117.164,421.735,172.018,30.405,155.638
C04424=1060.428,116.915,421.755,172.016,30.402,155.637
C04425=1060.423,116.666,421.776,172.014,30.400,155.637
C04426=1060.417,116.417,421.795,172.012,30.397,155.636
C04427=1060.411,116.167,421.815,172.011,30.394,155.636
C04428=1060.405,115.919,421.835,172.009,30.392,155.636
C04429=1060.399,115.669,421.855,172.008,30.389,155.635
C04430=1060.394,115.420,421.875,172.006,30.386,155.635
C04431=1060.388,115.171,421.895,172.004,30.384,155.634
C04432=1060.382,114.922,421.914,172.003,30.380,155.634
C04433=1060.376,114.673,421.934,172.001,30.378,155.633
C04434=1060.371,114.424,421.954,171.999,30.375,155.633
C04435=1060.365,114.175,421.974,171.998,30.373,155.633
C04436=1060.359,113.926,421.994,171.997,30.370,155.632
C04437=1060.354,113.676,422.013,171.995,30.368,155.632
C04438=1060.347,113.428,422.033,171.993,30.365,155.631
C04439=1060.341,113.178,422.052,171.991,30.362,155.631
C04440=1060.335,112.929,422.072,171.990,30.360,155.631
C04441=1060.329,112.679,422.092,171.988,30.357,155.630
C04442=1060.323,112.430,422.111,171.987,30.354,155.630
C04443=1060.317,112.181,422.131,171.985,30.352,155.629
C04444=1060.311,111.932,422.151,171.984,30.349,155.629
C04445=1060.306,111.683,422.170,171.982,30.346,155.629
C04446=1060.300,111.434,422.190,171.980,30.344,155.628
C04447=1060.294,111.185,422.209,171.978,30.341,155.628
C04448=1060.288,110.936,422.229,171.977,30.338,155.627
C04449=1060.281,110.651,422.251,171.975,30.336,155.627
C04450=1060.274,110.366,422.274,171.973,30.333,155.627
C04451=1060.267,110.081,422.296,171.971,30.330,155.626
C04452=1060.260,109.797,422.318,171.970,30.327,155.626
C04453=1060.254,109.548,422.338,171.968,30.324,155.625
C04454=1060.248,109.298,422.357,171.967,30.322,155.625
C04455=1060.242,109.049,422.377,171.965,30.319,155.624
C04456=1060.236,108.800,422.396,171.963,30.316,155.624
C04457=1060.230,108.551,422.415,171.962,30.314,155.624
C04458=1060.224,108.302,422.435,171.960,30.311,155.623
C04459=1060.219,108.053,422.454,171.958,30.309,155.623
C04460=1060.213,107.804,422.474,171.957,30.306,155.622
C04461=1060.206,107.555,422.493,171.956,30.304,155.622
C04462=1060.201,107.305,422.512,171.954,30.301,155.622
C04463=1060.195,107.056,422.532,171.952,30.298,155.621
C04464=1060.189,106.807,422.551,171.950,30.296,155.621
C04465=1060.183,106.558,422.570,171.949,30.293,155.620
C04466=1060.176,106.309,422.590,171.948,30.290,155.620
C04467=1060.171,106.060,422.609,171.946,30.288,155.620
C04468=1060.165,105.810,422.628,171.944,30.285,155.619
C04469=1060.159,105.561,422.648,171.943,30.283,155.619
C04470=1060.153,105.312,422.667,171.941,30.280,155.618
C04471=1060.147,105.063,422.686,171.940,30.278,155.618
C04472=1060.141,104.813,422.705,171.938,30.275,155.618
C04473=1060.135,104.565,422.725,171.937,30.272,155.617
C04474=1060.130,104.315,422.744,171.935,30.269,155.617
C04475=1060.123,104.066,422.763,171.933,30.267,155.616
C04476=1060.118,103.817,422.782,171.931,30.264,155.616
C04477=1060.112,103.568,422.802,171.930,30.262,155.616
C04478=1060.106,103.318,422.822,171.929,30.259,155.615
C04479=1060.099,103.069,422.840,171.927,30.256,155.615
C04480=1060.094,102.820,422.859,171.925,30.254,155.614
C04481=1060.088,102.570,422.879,171.923,30.251,155.614
C04482=1060.083,102.322,422.898,171.923,30.249,155.614
C04483=1060.076,102.073,422.917,171.921,30.246,155.613
C04484=1060.071,101.824,422.936,171.919,30.243,155.613
C04485=1060.065,101.574,422.955,171.917,30.241,155.612
C04486=1060.059,101.325,422.975,171.916,30.238,155.612
C04487=1060.053,101.075,422.994,171.915,30.235,155.612
C04488=1060.047,100.826,423.013,171.913,30.233,155.611
C04489=1060.041,100.577,423.032,171.911,30.230,155.611
C04490=1060.035,100.328,423.051,171.910,30.227,155.610
C04491=1060.029,100.079,423.070,171.908,30.225,155.610
C04492=1060.023,99.830,423.089,171.907,30.223,155.610
C04493=1060.017,99.580,423.108,171.905,30.220,155.609
C04494=1060.010,99.331,423.127,171.904,30.217,155.609
C04495=1060.005,99.082,423.146,171.902,30.215,155.608
C04496=1059.998,98.833,423.165,171.900,30.212,155.608
C04497=1059.993,98.584,423.184,171.899,30.210,155.608
C04498=1059.987,98.335,423.202,171.898,30.207,155.607
C04499=1059.981,98.085,423.222,171.896,30.204,155.607
C04500=1059.975,97.836,423.240,171.894,30.202,155.606
C04501=1059.969,97.587,423.259,171.892,30.199,155.606
C04502=1059.963,97.337,423.279,171.892,30.197,155.606
C04503=1059.957,97.088,423.297,171.890,30.194,155.605
C04504=1059.951,96.839,423.317,171.888,30.192,155.605
C04505=1059.945,96.590,423.335,171.886,30.189,155.605
C04506=1059.939,96.340,423.354,171.884,30.186,155.604
C04507=1059.933,96.092,423.373,171.884,30.184,155.604
C04508=1059.928,95.842,423.392,171.882,30.181,155.603
C04509=1059.921,95.593,423.411,171.880,30.178,155.603
C04510=1059.915,95.344,423.429,171.878,30.176,155.603
C04511=1059.909,95.095,423.449,171.877,30.174,155.602
C04512=1059.903,94.845,423.466,171.876,30.171,155.602
C04513=1059.897,94.561,423.488,171.874,30.168,155.601
C04514=1059.890,94.276,423.510,171.872,30.165,155.601
C04515=1059.883,93.992,423.531,171.870,30.162,155.600
C04516=1059.876,93.707,423.553,171.868,30.159,155.600
C04517=1059.870,93.458,423.571,171.867,30.156,155.600
C04518=1059.864,93.209,423.591,171.866,30.154,155.599
C04519=1059.858,92.960,423.609,171.864,30.151,155.599
C04520=1059.853,92.710,423.628,171.862,30.149,155.598
C04521=1059.846,92.461,423.646,171.861,30.146,155.598
C04522=1059.841,92.212,423.665,171.860,30.143,155.598
C04523=1059.835,91.963,423.684,171.858,30.141,155.597
C04524=1059.829,91.713,423.703,171.856,30.138,155.597
C04525=1059.823,91.464,423.721,171.854,30.135,155.596
C04526=1059.817,91.214,423.740,171.854,30.133,155.596
C04527=1059.811,90.966,423.759,171.852,30.130,155.596
C04528=1059.805,90.717,423.777,171.850,30.127,155.595
C04529=1059.799,90.467,423.797,171.848,30.125,155.595
C04530=1059.793,90.217,423.814,171.847,30.123,155.594
C04531=1059.787,89.968,423.833,171.846,30.120,155.594
C04532=1059.781,89.720,423.851,171.844,30.117,155.594
C04533=1059.776,89.470,423.870,171.842,30.115,155.593
C04534=1059.769,89.221,423.889,171.841,30.112,155.593
C04535=1059.763,88.972,423.907,171.840,30.110,155.592
C04536=1059.756,88.722,423.926,171.838,30.107,155.592
C04537=1059.751,88.473,423.944,171.836,30.105,155.592
C04538=1059.745,88.224,423.963,171.835,30.102,155.591
C04539=1059.739,87.975,423.981,171.833,30.100,155.591
C04540=1059.733,87.725,423.999,171.832,30.097,155.591
C04541=1059.726,87.476,424.018,171.830,30.094,155.590
C04542=1059.721,87.227,424.037,171.828,30.092,155.590
C04543=1059.715,86.978,424.055,171.827,30.090,155.589
C04544=1059.708,86.728,424.073,171.826,30.087,155.589
C04545=1059.702,86.479,424.091,171.824,30.084,155.589
C04546=1059.696,86.230,424.110,171.823,30.082,155.588
C04547=1059.691,85.981,424.129,171.821,30.079,155.588
C04548=1059.685,85.731,424.147,171.819,30.077,155.588
C04549=1059.678,85.482,424.165,171.818,30.074,155.587
C04550=1059.673,85.233,424.183,171.817,30.071,155.587
C04551=1059.666,84.984,424.202,171.815,30.069,155.586
C04552=1059.660,84.735,424.220,171.813,30.067,155.586
C04553=1059.655,84.485,424.239,171.812,30.064,155.586
C04554=1059.649,84.236,424.257,171.810,30.061,155.585
C04555=1059.643,83.986,424.275,171.809,30.059,155.585
C04556=1059.636,83.737,424.294,171.807,30.056,155.584
C04557=1059.631,83.488,424.311,171.805,30.053,155.584
C04558=1059.625,83.239,424.330,171.804,30.051,155.584
C04559=1059.619,82.989,424.348,171.803,30.049,155.583
C04560=1059.613,82.741,424.367,171.801,30.046,155.583
C04561=1059.607,82.491,424.385,171.799,30.043,155.582
C04562=1059.600,82.242,424.403,171.799,30.041,155.582
C04563=1059.595,81.993,424.421,171.797,30.038,155.582
C04564=1059.588,81.744,424.439,171.795,30.036,155.581
C04565=1059.583,81.494,424.458,171.793,30.033,155.581
C04566=1059.577,81.245,424.476,171.793,30.030,155.580
C04567=1059.571,80.995,424.494,171.791,30.028,155.580
C04568=1059.565,80.746,424.513,171.789,30.025,155.580
C04569=1059.559,80.497,424.530,171.787,30.022,155.579
C04570=1059.553,80.248,424.548,171.787,30.020,155.579
C04571=1059.547,79.998,424.568,171.785,30.018,155.579
C04572=1059.542,79.749,424.585,171.783,30.015,155.578
C04573=1059.535,79.500,424.604,171.781,30.012,155.578
C04574=1059.529,79.250,424.622,171.780,30.009,155.577
C04575=1059.524,79.001,424.639,171.779,30.007,155.577
C04576=1059.517,78.752,424.658,171.777,30.004,155.576
C04577=1059.511,78.467,424.678,171.775,30.001,155.576
C04578=1059.504,78.183,424.699,171.774,29.999,155.576
C04579=1059.497,77.899,424.720,171.772,29.995,155.575
C04580=1059.490,77.614,424.740,171.770,29.993,155.575
C04581=1059.484,77.365,424.758,171.769,29.990,155.574
C04582=1059.478,77.115,424.776,171.767,29.988,155.574
C04583=1059.472,76.866,424.794,171.766,29.985,155.574
C04584=1059.466,76.617,424.812,171.764,29.983,155.573
C04585=1059.460,76.367,424.830,171.763,29.980,155.573
C04586=1059.454,76.119,424.848,171.761,29.978,155.573
C04587=1059.448,75.869,424.866,171.760,29.975,155.572
C04588=1059.442,75.619,424.884,171.758,29.972,155.572
C04589=1059.437,75.370,424.902,171.757,29.970,155.571
C04590=1059.430,75.121,424.920,171.755,29.968,155.571
C04591=1059.423,74.871,424.938,171.753,29.965,155.571
C04592=1059.418,74.622,424.955,171.752,29.962,155.570
C04593=1059.412,74.373,424.973,171.751,29.960,155.570
C04594=1059.406,74.124,424.991,171.749,29.957,155.570
C04595=1059.400,73.875,425.009,171.747,29.955,155.569
C04596=1059.394,73.625,425.027,171.746,29.952,155.569
C04597=1059.388,73.376,425.045,171.745,29.949,155.568
C04598=1059.382,73.126,425.063,171.743,29.947,155.568
C04599=1059.376,72.878,425.081,171.741,29.945,155.568
C04600=1059.369,72.628,425.098,171.740,29.942,155.567
C04601=1059.364,72.379,425.116,171.739,29.939,155.567
C04602=1059.358,72.129,425.134,171.737,29.937,155.566
C04603=1059.352,71.880,425.151,171.735,29.934,155.566
C04604=1059.346,71.631,425.169,171.734,29.932,155.566
C04605=1059.340,71.382,425.187,171.733,29.929,155.565
C04606=1059.334,71.132,425.204,171.731,29.926,155.565
C04607=1059.327,70.883,425.223,171.729,29.924,155.564
C04608=1059.322,70.634,425.241,171.728,29.922,155.564
C04609=1059.315,70.384,425.258,171.727,29.919,155.564
C04610=1059.310,70.135,425.276,171.725,29.916,155.563
C04611=1059.304,69.885,425.294,171.723,29.914,155.563
C04612=1059.298,69.637,425.311,171.723,29.912,155.563
C04613=1059.291,69.387,425.329,171.721,29.909,155.562
C04614=1059.286,69.138,425.346,171.719,29.906,155.562
C04615=1059.280,68.888,425.364,171.717,29.903,155.561
C04616=1059.274,68.639,425.381,171.716,29.901,155.561
C04617=1059.267,68.390,425.399,171.715,29.899,155.561
C04618=1059.262,68.141,425.417,171.713,29.896,155.560
C04619=1059.256,67.891,425.435,171.711,29.894,155.560
C04620=1059.250,67.642,425.452,171.710,29.891,155.560
C04621=1059.243,67.392,425.470,171.709,29.889,155.559
C04622=1059.238,67.143,425.487,171.707,29.886,155.559
C04623=1059.231,66.894,425.505,171.705,29.884,155.559
C04624=1059.226,66.645,425.522,171.704,29.881,155.558
C04625=1059.219,66.395,425.540,171.703,29.878,155.558
C04626=1059.213,66.146,425.557,171.701,29.876,155.557
C04627=1059.207,65.897,425.575,171.699,29.874,155.557
C04628=1059.202,65.648,425.593,171.698,29.871,155.557
C04629=1059.195,65.398,425.610,171.697,29.868,155.556
C04630=1059.189,65.149,425.627,171.695,29.866,155.556
C04631=1059.183,64.899,425.645,171.694,29.863,155.555
C04632=1059.177,64.650,425.662,171.692,29.861,155.555
C04633=1059.171,64.400,425.680,171.691,29.858,155.555
C04634=1059.165,64.152,425.697,171.689,29.856,155.554
C04635=1059.159,63.902,425.714,171.688,29.853,155.554
C04636=1059.152,63.653,425.731,171.686,29.851,155.554
C04637=1059.146,63.403,425.749,171.685,29.849,155.553
C04638=1059.140,63.155,425.766,171.683,29.846,155.553
C04639=1059.134,62.904,425.784,171.682,29.844,155.553
C04640=1059.128,62.656,425.801,171.680,29.841,155.552
C04641=1059.120,62.371,425.820,171.678,29.838,155.552
C04642=1059.114,62.086,425.840,171.676,29.835,155.551
C04643=1059.106,61.801,425.860,171.675,29.833,155.551
C04644=1059.099,61.517,425.880,171.673,29.830,155.551
C04645=1059.093,61.267,425.896,171.671,29.827,155.550
C04646=1059.087,61.018,425.914,171.671,29.825,155.550
C04647=1059.081,60.769,425.931,171.669,29.822,155.549
C04648=1059.075,60.520,425.948,171.667,29.820,155.549
C04649=1059.069,60.270,425.966,171.665,29.818,155.549
C04650=1059.063,60.021,425.983,171.665,29.815,155.548
C04651=1059.056,59.771,426.000,171.663,29.812,155.548
C04652=1059.051,59.522,426.017,171.661,29.810,155.548
C04653=1059.044,59.272,426.034,171.659,29.807,155.547
C04654=1059.038,59.023,426.052,171.659,29.805,155.547
C04655=1059.031,58.774,426.069,171.657,29.803,155.547
C04656=1059.026,58.525,426.085,171.655,29.800,155.546
C04657=1059.020,58.276,426.103,171.653,29.798,155.546
C04658=1059.013,58.026,426.120,171.652,29.795,155.546
C04659=1059.008,57.776,426.137,171.651,29.793,155.545
C04660=1059.001,57.527,426.154,171.649,29.790,155.545
C04661=1058.995,57.278,426.171,171.648,29.788,155.544
C04662=1058.990,57.029,426.188,171.646,29.785,155.544
C04663=1058.983,56.779,426.205,171.645,29.783,155.544
C04664=1058.977,56.530,426.222,171.643,29.780,155.543
C04665=1058.971,56.281,426.239,171.642,29.777,155.543
C04666=1058.964,56.031,426.257,171.640,29.775,155.543
C04667=1058.958,55.782,426.273,171.639,29.773,155.542
C04668=1058.952,55.532,426.291,171.637,29.771,155.542
C04669=1058.946,55.283,426.307,171.636,29.768,155.542
C04670=1058.941,55.034,426.325,171.634,29.765,155.541
C04671=1058.934,54.784,426.342,171.633,29.763,155.541
C04672=1058.928,54.535,426.358,171.631,29.760,155.540
C04673=1058.923,54.286,426.376,171.630,29.758,155.540
C04674=1058.916,54.036,426.392,171.628,29.755,155.540
C04675=1058.910,53.787,426.409,171.627,29.753,155.539
C04676=1058.905,53.538,426.426,171.626,29.750,155.539
C04677=1058.898,53.288,426.444,171.624,29.748,155.539
C04678=1058.892,53.039,426.460,171.622,29.745,155.538
C04679=1058.886,52.790,426.477,171.621,29.743,155.538
C04680=1058.880,52.540,426.494,171.620,29.741,155.537
C04681=1058.873,52.291,426.511,171.618,29.738,155.537
C04682=1058.868,52.041,426.528,171.616,29.735,155.537
C04683=1058.862,51.793,426.545,171.615,29.733,155.536
C04684=1058.855,51.543,426.561,171.614,29.730,155.536
C04685=1058.850,51.294,426.579,171.612,29.728,155.536
C04686=1058.844,51.044,426.595,171.610,29.725,155.535
C04687=1058.838,50.795,426.612,171.608,29.723,155.535
C04688=1058.832,50.545,426.629,171.608,29.720,155.534
C04689=1058.826,50.296,426.646,171.606,29.718,155.534
C04690=1058.820,50.047,426.663,171.604,29.715,155.534
C04691=1058.814,49.798,426.679,171.603,29.713,155.533
C04692=1058.808,49.548,426.697,171.602,29.711,155.533
C04693=1058.802,49.299,426.713,171.600,29.708,155.533
C04694=1058.795,49.050,426.730,171.598,29.705,155.532
C04695=1058.790,48.800,426.747,171.597,29.703,155.532
C04696=1058.784,48.550,426.764,171.596,29.700,155.532
C04697=1058.777,48.301,426.781,171.594,29.698,155.531
C04698=1058.772,48.052,426.797,171.592,29.695,155.531
C04699=1058.766,47.802,426.814,171.591,29.693,155.531
C04700=1058.759,47.553,426.831,171.590,29.690,155.530
C04701=1058.753,47.304,426.847,171.588,29.688,155.530
C04702=1058.748,47.055,426.865,171.587,29.685,155.529
C04703=1058.742,46.805,426.881,171.585,29.682,155.529
C04704=1058.736,46.556,426.897,171.584,29.680,155.529
C04705=1058.730,46.271,426.917,171.582,29.677,155.528
C04706=1058.722,45.986,426.936,171.581,29.674,155.528
C04707=1058.715,45.701,426.955,171.579,29.672,155.527
C04708=1058.708,45.416,426.974,171.577,29.669,155.527
C04709=1058.703,45.166,426.991,171.576,29.666,155.527
C04710=1058.697,44.917,427.007,171.574,29.663,155.526
C04711=1058.691,44.668,427.024,171.572,29.661,155.526
C04712=1058.684,44.418,427.041,171.571,29.659,155.526
C04713=1058.679,44.169,427.057,171.570,29.656,155.525
C04714=1058.673,43.919,427.074,171.568,29.653,155.525
C04715=1058.667,43.670,427.090,171.566,29.651,155.524
C04716=1058.661,43.421,427.107,171.566,29.648,155.524
C04717=1058.655,43.172,427.123,171.564,29.646,155.524
C04718=1058.648,42.922,427.140,171.562,29.644,155.523
C04719=1058.642,42.672,427.156,171.560,29.641,155.523
C04720=1058.636,42.423,427.172,171.560,29.639,155.523
C04721=1058.631,42.174,427.190,171.558,29.636,155.522
C04722=1058.625,41.925,427.206,171.556,29.634,155.522
C04723=1058.618,41.675,427.223,171.555,29.631,155.522
C04724=1058.613,41.425,427.239,171.553,29.628,155.521
C04725=1058.607,41.176,427.255,171.552,29.626,155.521
C04726=1058.601,40.927,427.272,171.550,29.624,155.520
C04727=1058.595,40.677,427.288,171.549,29.621,155.520
C04728=1058.589,40.428,427.304,171.547,29.619,155.520
C04729=1058.582,40.179,427.321,171.546,29.617,155.519
C04730=1058.576,39.929,427.338,171.544,29.614,155.519
C04731=1058.570,39.680,427.354,171.543,29.611,155.519
C04732=1058.564,39.430,427.370,171.541,29.609,155.518
C04733=1058.558,39.181,427.386,171.540,29.607,155.518
C04734=1058.552,38.932,427.403,171.539,29.604,155.518
C04735=1058.546,38.682,427.419,171.537,29.602,155.517
C04736=1058.540,38.433,427.435,171.535,29.599,155.517
C04737=1058.534,38.184,427.451,171.534,29.597,155.517
C04738=1058.528,37.934,427.468,171.533,29.594,155.516
C04739=1058.522,37.684,427.484,171.531,29.592,155.516
C04740=1058.516,37.435,427.501,171.529,29.589,155.516
C04741=1058.509,37.186,427.516,171.528,29.587,155.515
C04742=1058.503,36.936,427.532,171.527,29.584,155.515
C04743=1058.497,36.687,427.549,171.525,29.582,155.515
C04744=1058.491,36.438,427.565,171.523,29.580,155.514
C04745=1058.485,36.188,427.581,171.522,29.577,155.514
C04746=1058.479,35.939,427.598,171.521,29.575,155.513
C04747=1058.472,35.689,427.614,171.519,29.573,155.513
C04748=1058.466,35.440,427.630,171.517,29.570,155.513
C04749=1058.460,35.191,427.646,171.516,29.568,155.512
C04750=1058.454,34.941,427.662,171.514,29.565,155.512
C04751=1058.448,34.692,427.679,171.513,29.563,155.512
C04752=1058.442,34.442,427.694,171.512,29.560,155.511
C04753=1058.436,34.193,427.710,171.510,29.558,155.511
C04754=1058.430,33.944,427.726,171.508,29.555,155.511
C04755=1058.424,33.694,427.742,171.507,29.553,155.510
C04756=1058.418,33.445,427.759,171.506,29.551,155.510
C04757=1058.411,33.196,427.774,171.504,29.548,155.510
C04758=1058.405,32.947,427.790,171.502,29.546,155.509
C04759=1058.399,32.697,427.807,171.500,29.543,155.509
C04760=1058.393,32.446,427.823,171.500,29.541,155.509
C04761=1058.387,32.197,427.838,171.498,29.539,155.508
C04762=1058.381,31.948,427.855,171.496,29.536,155.508
C04763=1058.375,31.699,427.871,171.495,29.534,155.508
C04764=1058.369,31.449,427.887,171.494,29.532,155.507
C04765=1058.363,31.200,427.903,171.492,29.529,155.507
C04766=1058.356,30.950,427.918,171.490,29.527,155.507
C04767=1058.350,30.701,427.935,171.489,29.524,155.506
C04768=1058.344,30.452,427.951,171.487,29.522,155.506
C04769=1058.336,30.105,427.973,171.485,29.519,155.506
C04770=1058.328,29.758,427.995,171.483,29.515,155.505
C04771=1058.319,29.411,428.017,171.481,29.512,155.505
C04772=1058.311,29.064,428.039,171.479,29.508,155.504
C04773=1058.305,28.815,428.056,171.478,29.506,155.504
C04774=1058.299,28.565,428.070,171.476,29.503,155.503
C04775=1058.293,28.316,428.087,171.474,29.501,155.503
C04776=1058.287,28.067,428.103,171.473,29.498,155.503
C04777=1058.280,27.817,428.118,171.472,29.496,155.502
C04778=1058.274,27.568,428.134,171.470,29.494,155.502
C04779=1058.268,27.319,428.150,171.468,29.491,155.502
C04780=1058.262,27.069,428.166,171.467,29.489,155.501
C04781=1058.256,26.819,428.182,171.465,29.487,155.501
C04782=1058.249,26.570,428.197,171.464,29.485,155.501
C04783=1058.244,26.320,428.213,171.463,29.482,155.500
C04784=1058.237,26.071,428.229,171.461,29.480,155.500
C04785=1058.231,25.822,428.245,171.459,29.477,155.500
C04786=1058.225,25.572,428.260,171.457,29.475,155.499
C04787=1058.219,25.323,428.276,171.457,29.473,155.499
C04788=1058.213,25.073,428.292,171.455,29.470,155.499
C04789=1058.207,24.824,428.307,171.453,29.468,155.498
C04790=1058.201,24.574,428.323,171.451,29.466,155.498
C04791=1058.194,24.325,428.338,171.451,29.463,155.498
C04792=1058.188,24.075,428.355,171.449,29.461,155.497
C04793=1058.182,23.826,428.370,171.447,29.458,155.497
C04794=1058.176,23.576,428.386,171.446,29.456,155.497
C04795=1058.169,23.327,428.402,171.444,29.454,155.496
C04796=1058.164,23.078,428.417,171.443,29.451,155.496
C04797=1058.157,22.829,428.432,171.441,29.449,155.496
C04798=1058.152,22.579,428.448,171.440,29.446,155.495
C04799=1058.145,22.330,428.464,171.438,29.444,155.495
C04800=1058.139,22.080,428.479,171.436,29.442,155.495
C04801=1058.134,21.831,428.495,171.436,29.439,155.494
C04802=1058.127,21.581,428.510,171.434,29.437,155.494
C04803=1058.121,21.332,428.527,171.432,29.434,155.494
C04804=1058.115,21.082,428.541,171.430,29.432,155.493
C04805=1058.109,20.833,428.558,171.429,29.430,155.493
C04806=1058.103,20.584,428.572,171.428,29.427,155.493
C04807=1058.097,20.334,428.588,171.426,29.425,155.493
C04808=1058.091,20.085,428.604,171.425,29.422,155.492
C04809=1058.085,19.866,428.617,171.423,29.421,155.492
C04810=1058.080,19.647,428.630,171.422,29.419,155.492
C04811=1058.074,19.430,428.644,171.420,29.417,155.491
C04812=1058.069,19.211,428.658,171.419,29.415,155.491
C04813=1058.063,18.992,428.671,171.418,29.412,155.491
C04814=1058.058,18.773,428.685,171.417,29.410,155.490
C04815=1058.053,18.555,428.698,171.415,29.408,155.490
C04816=1058.047,18.337,428.712,171.413,29.406,155.490
C04817=1058.041,18.087,428.727,171.413,29.404,155.490
C04818=1058.035,17.837,428.742,171.411,29.401,155.489
C04819=1058.030,17.589,428.758,171.409,29.399,155.489
C04820=1058.023,17.339,428.773,171.408,29.397,155.489
C04821=1058.017,17.089,428.788,171.406,29.394,155.488
C04822=1058.011,16.840,428.804,171.405,29.392,155.488
C04823=1058.005,16.590,428.819,171.403,29.390,155.488
C04824=1057.999,16.340,428.835,171.402,29.387,155.487
C04825=1057.992,16.091,428.850,171.400,29.385,155.487
C04826=1057.986,15.842,428.865,171.398,29.383,155.487
C04827=1057.981,15.592,428.881,171.397,29.380,155.486
C04828=1057.974,15.343,428.896,171.396,29.378,155.486
C04829=1057.968,15.094,428.911,171.394,29.376,155.486
C04830=1057.962,14.844,428.927,171.392,29.373,155.485
C04831=1057.956,14.595,428.941,171.391,29.371,155.485
C04832=1057.950,14.346,428.957,171.389,29.369,155.485
C04833=1057.943,14.061,428.974,171.387,29.366,155.484
C04834=1057.936,13.778,428.992,171.386,29.364,155.484
C04835=1057.928,13.494,429.009,171.384,29.361,155.484
C04836=1057.922,13.211,429.026,171.382,29.358,155.483
C04837=1057.915,12.961,429.041,171.380,29.356,155.483
C04838=1057.909,12.711,429.056,171.379,29.354,155.483
C04839=1057.903,12.462,429.071,171.378,29.352,155.483
C04840=1057.896,12.212,429.086,171.376,29.350,155.482
C04841=1057.890,11.964,429.101,171.375,29.347,155.482
C04842=1057.884,11.714,429.117,171.373,29.345,155.482
C04843=1057.878,11.464,429.132,171.371,29.343,155.481
C04844=1057.872,11.214,429.147,171.370,29.341,155.481
C04845=1057.865,10.965,429.162,171.369,29.338,155.481
C04846=1057.860,10.716,429.176,171.367,29.336,155.480
C04847=1057.853,10.466,429.191,171.365,29.333,155.480
C04848=1057.847,10.216,429.206,171.364,29.331,155.480
C04849=1057.840,9.967,429.222,171.362,29.329,155.480
C04850=1057.834,9.718,429.237,171.361,29.327,155.479
C04851=1057.829,9.468,429.252,171.359,29.324,155.479
C04852=1057.822,9.219,429.267,171.358,29.322,155.479
C04853=1057.816,8.969,429.282,171.356,29.320,155.478
C04854=1057.810,8.719,429.297,171.354,29.318,155.478
C04855=1057.804,8.471,429.311,171.352,29.316,155.478
C04856=1057.797,8.221,429.326,171.352,29.313,155.477
C04857=1057.791,7.971,429.341,171.350,29.311,155.477
C04858=1057.785,7.722,429.356,171.348,29.309,155.477
C04859=1057.779,7.473,429.371,171.347,29.306,155.476
C04860=1057.772,7.223,429.386,171.345,29.304,155.476
C04861=1057.767,6.973,429.401,171.343,29.302,155.476
C04862=1057.761,6.724,429.416,171.342,29.299,155.475
C04863=1057.755,6.474,429.431,171.341,29.297,155.475
C04864=1057.748,6.225,429.446,171.339,29.295,155.475
C04865=1057.742,5.975,429.461,171.337,29.293,155.475
C04866=1057.736,5.726,429.475,171.335,29.291,155.474
C04867=1057.730,5.476,429.490,171.334,29.288,155.474
C04868=1057.723,5.227,429.505,171.333,29.286,155.474
C04869=1057.718,4.978,429.520,171.331,29.284,155.473
C04870=1057.711,4.728,429.535,171.330,29.282,155.473
C04871=1057.705,4.479,429.550,171.328,29.279,155.473
C04872=1057.699,4.230,429.564,171.326,29.277,155.472
C04873=1057.693,3.980,429.579,171.324,29.274,155.472
C04874=1057.687,3.730,429.595,171.324,29.272,155.472
C04875=1057.681,3.481,429.609,171.322,29.270,155.472
C04876=1057.675,3.231,429.624,171.320,29.268,155.471
C04877=1057.669,2.981,429.638,171.319,29.266,155.471
C04878=1057.663,2.732,429.653,171.317,29.263,155.471
C04879=1057.657,2.482,429.668,171.315,29.261,155.470
C04880=1057.650,2.233,429.683,171.313,29.259,155.470
C04881=1057.644,1.984,429.698,171.313,29.257,155.470
C04882=1057.638,1.734,429.712,171.311,29.254,155.470
C04883=1057.632,1.485,429.727,171.309,29.252,155.469
C04884=1057.626,1.235,429.741,171.308,29.249,155.469
C04885=1057.620,0.985,429.756,171.306,29.247,155.469
C04886=1057.614,0.736,429.771,171.304,29.245,155.468
C04887=1057.608,0.487,429.786,171.303,29.243,155.468
C04888=1057.602,0.238,429.800,171.302,29.241,155.468
C04889=1057.595,-0.012,429.815,171.300,29.239,155.468
C04890=1057.589,-0.262,429.830,171.298,29.236,155.467
C04891=1057.584,-0.511,429.844,171.297,29.234,155.467
C04892=1057.577,-0.761,429.859,171.295,29.231,155.467
C04893=1057.571,-1.010,429.874,171.293,29.229,155.466
C04894=1057.565,-1.260,429.888,171.292,29.227,155.466
C04895=1057.560,-1.509,429.902,171.291,29.225,155.466
C04896=1057.553,-1.759,429.917,171.289,29.222,155.465
C04897=1057.546,-2.041,429.934,171.287,29.220,155.465
C04898=1057.540,-2.322,429.950,171.286,29.217,155.465
C04899=1057.533,-2.604,429.967,171.284,29.215,155.464
C04900=1057.526,-2.886,429.983,171.282,29.212,155.464
C04901=1057.520,-3.135,429.998,171.280,29.210,155.464
C04902=1057.514,-3.385,430.012,171.279,29.208,155.463
C04903=1057.508,-3.634,430.027,171.277,29.206,155.463
C04904=1057.502,-3.884,430.042,171.275,29.204,155.463
C04905=1057.495,-4.134,430.055,171.274,29.201,155.463
C04906=1057.489,-4.383,430.070,171.272,29.199,155.462
C04907=1057.483,-4.633,430.085,171.270,29.197,155.462
C04908=1057.477,-4.882,430.098,171.269,29.195,155.462
C04909=1057.470,-5.132,430.113,171.268,29.193,155.462
C04910=1057.464,-5.381,430.128,171.266,29.191,155.461
C04911=1057.458,-5.631,430.142,171.264,29.188,155.461
C04912=1057.451,-5.880,430.156,171.263,29.186,155.461
C04913=1057.446,-6.130,430.170,171.261,29.184,155.460
C04914=1057.439,-6.379,430.185,171.259,29.182,155.460
C04915=1057.433,-6.629,430.198,171.257,29.180,155.460
C04916=1057.427,-6.878,430.213,171.257,29.178,155.460
C04917=1057.421,-7.127,430.228,171.255,29.175,155.459
C04918=1057.415,-7.378,430.242,171.253,29.173,155.459
C04919=1057.408,-7.626,430.256,171.251,29.171,155.459
C04920=1057.402,-7.876,430.270,171.250,29.169,155.459
C04921=1057.396,-8.126,430.285,171.248,29.167,155.458
C04922=1057.390,-8.375,430.298,171.246,29.164,155.458
C04923=1057.383,-8.625,430.313,171.245,29.162,155.458
C04924=1057.378,-8.875,430.327,171.244,29.161,155.458
C04925=1057.371,-9.124,430.342,171.242,29.159,155.457
C04926=1057.365,-9.374,430.355,171.240,29.156,155.457
C04927=1057.359,-9.623,430.370,171.239,29.154,155.457
C04928=1057.353,-9.873,430.384,171.237,29.152,155.456
C04929=1057.347,-10.121,430.398,171.235,29.150,155.456
C04930=1057.341,-10.372,430.412,171.233,29.148,155.456
C04931=1057.335,-10.621,430.427,171.232,29.145,155.456
C04932=1057.328,-10.871,430.441,171.230,29.143,155.455
C04933=1057.323,-11.120,430.455,171.229,29.141,155.455
C04934=1057.316,-11.370,430.469,171.228,29.139,155.455
C04935=1057.310,-11.619,430.483,171.226,29.137,155.454
C04936=1057.304,-11.869,430.498,171.224,29.135,155.454
C04937=1057.298,-12.118,430.512,171.222,29.132,155.454
C04938=1057.292,-12.368,430.525,171.221,29.130,155.454
C04939=1057.286,-12.617,430.540,171.219,29.128,155.453
C04940=1057.280,-12.866,430.553,171.217,29.126,155.453
C04941=1057.273,-13.116,430.568,171.217,29.124,155.453
C04942=1057.268,-13.366,430.582,171.215,29.121,155.453
C04943=1057.261,-13.616,430.595,171.213,29.120,155.452
C04944=1057.255,-13.865,430.610,171.211,29.118,155.452
C04945=1057.250,-14.114,430.624,171.210,29.115,155.452
C04946=1057.243,-14.364,430.638,171.208,29.113,155.452
C04947=1057.237,-14.613,430.652,171.206,29.111,155.451
C04948=1057.231,-14.863,430.666,171.204,29.109,155.451
C04949=1057.225,-15.113,430.680,171.203,29.107,155.451
C04950=1057.219,-15.362,430.693,171.201,29.104,155.451
C04951=1057.212,-15.612,430.708,171.200,29.102,155.450
C04952=1057.207,-15.861,430.722,171.198,29.101,155.450
C04953=1057.200,-16.111,430.735,171.197,29.099,155.450
C04954=1057.193,-16.360,430.749,171.195,29.096,155.449
C04955=1057.187,-16.610,430.764,171.193,29.094,155.449
C04956=1057.181,-16.859,430.777,171.192,29.093,155.449
C04957=1057.176,-17.109,430.791,171.190,29.090,155.449
C04958=1057.169,-17.359,430.804,171.188,29.088,155.449
C04959=1057.162,-17.608,430.818,171.186,29.086,155.448
C04960=1057.156,-17.858,430.833,171.185,29.084,155.448
C04961=1057.149,-18.138,430.847,171.183,29.082,155.448
C04962=1057.142,-18.418,430.863,171.181,29.079,155.447
C04963=1057.135,-18.698,430.878,171.180,29.077,155.447
C04964=1057.128,-18.979,430.894,171.178,29.075,155.447
C04965=1057.122,-19.227,430.908,171.176,29.073,155.447
C04966=1057.116,-19.477,430.922,171.174,29.071,155.446
C04967=1057.110,-19.727,430.935,171.173,29.069,155.446
C04968=1057.104,-19.977,430.949,171.171,29.067,155.446
C04969=1057.098,-20.226,430.963,171.169,29.064,155.446
C04970=1057.091,-20.476,430.976,171.168,29.062,155.445
C04971=1057.086,-20.725,430.990,171.166,29.061,155.445
C04972=1057.079,-20.974,431.004,171.164,29.058,155.445
C04973=1057.073,-21.224,431.018,171.162,29.056,155.445
C04974=1057.067,-21.474,431.032,171.162,29.054,155.444
C04975=1057.061,-21.723,431.045,171.160,29.053,155.444
C04976=1057.055,-21.973,431.059,171.158,29.050,155.444
C04977=1057.048,-22.222,431.072,171.156,29.048,155.444
C04978=1057.042,-22.472,431.086,171.155,29.046,155.443
C04979=1057.036,-22.722,431.100,171.153,29.044,155.443
C04980=1057.030,-22.971,431.113,171.151,29.042,155.443
C04981=1057.024,-23.221,431.127,171.149,29.040,155.443
C04982=1057.017,-23.471,431.141,171.148,29.038,155.442
C04983=1057.011,-23.720,431.154,171.146,29.036,155.442
C04984=1057.006,-23.970,431.168,171.144,29.034,155.442
C04985=1057.000,-24.219,431.181,171.143,29.032,155.442
C04986=1056.993,-24.469,431.195,171.141,29.030,155.442
C04987=1056.987,-24.718,431.208,171.140,29.028,155.441
C04988=1056.981,-24.968,431.222,171.138,29.026,155.441
C04989=1056.975,-25.217,431.235,171.137,29.024,155.441
C04990=1056.969,-25.467,431.249,171.135,29.022,155.441
C04991=1056.963,-25.716,431.263,171.133,29.020,155.440
C04992=1056.956,-25.966,431.276,171.131,29.018,155.440
C04993=1056.951,-26.215,431.290,171.130,29.015,155.440
C04994=1056.944,-26.465,431.303,171.128,29.014,155.440
C04995=1056.938,-26.714,431.317,171.126,29.012,155.439
C04996=1056.932,-26.964,431.330,171.125,29.009,155.439
C04997=1056.926,-27.213,431.344,171.123,29.008,155.439
C04998=1056.920,-27.464,431.357,171.121,29.006,155.439
C04999=1056.913,-27.713,431.370,171.119,29.004,155.439
C05000=1056.907,-27.962,431.383,171.118,29.002,155.438
C05001=1056.901,-28.212,431.396,171.116,29.000,155.438
C05002=1056.894,-28.462,431.410,171.114,28.998,155.438
C05003=1056.889,-28.711,431.424,171.112,28.996,155.438
C05004=1056.883,-28.961,431.437,171.112,28.994,155.437
C05005=1056.877,-29.210,431.450,171.110,28.992,155.437
C05006=1056.870,-29.460,431.463,171.108,28.990,155.437
C05007=1056.864,-29.710,431.477,171.106,28.988,155.437
C05008=1056.857,-29.959,431.490,171.105,28.987,155.437
C05009=1056.851,-30.208,431.503,171.103,28.984,155.436
C05010=1056.845,-30.458,431.516,171.101,28.983,155.436
C05011=1056.838,-30.708,431.529,171.099,28.981,155.436
C05012=1056.832,-30.957,431.543,171.098,28.979,155.436
C05013=1056.827,-31.207,431.557,171.096,28.977,155.435
C05014=1056.821,-31.456,431.570,171.094,28.974,155.435
C05015=1056.815,-31.706,431.582,171.092,28.973,155.435
C05016=1056.808,-31.956,431.596,171.091,28.971,155.435
C05017=1056.802,-32.205,431.609,171.089,28.969,155.435
C05018=1056.795,-32.454,431.623,171.087,28.967,155.434
C05019=1056.789,-32.704,431.635,171.086,28.965,155.434
C05020=1056.783,-32.954,431.648,171.084,28.963,155.434
C05021=1056.777,-33.203,431.662,171.082,28.961,155.434
C05022=1056.771,-33.453,431.675,171.080,28.959,155.434
C05023=1056.764,-33.703,431.688,171.079,28.957,155.433
C05024=1056.758,-33.952,431.701,171.077,28.955,155.433
C05025=1056.752,-34.231,431.715,171.075,28.954,155.433
C05026=1056.745,-34.511,431.730,171.073,28.951,155.433
C05027=1056.738,-34.790,431.745,171.072,28.949,155.432
C05028=1056.731,-35.070,431.760,171.070,28.947,155.432
C05029=1056.725,-35.319,431.773,171.068,28.945,155.432
C05030=1056.719,-35.569,431.786,171.067,28.943,155.432
C05031=1056.712,-35.819,431.799,171.065,28.942,155.432
C05032=1056.706,-36.069,431.812,171.063,28.939,155.431
C05033=1056.700,-36.318,431.825,171.061,28.938,155.431
C05034=1056.694,-36.567,431.838,171.060,28.935,155.431
C05035=1056.688,-36.817,431.851,171.058,28.934,155.431
C05036=1056.682,-37.066,431.864,171.056,28.932,155.430
C05037=1056.676,-37.316,431.877,171.054,28.930,155.430
C05038=1056.670,-37.565,431.890,171.053,28.928,155.430
C05039=1056.664,-37.815,431.903,171.051,28.926,155.430
C05040=1056.658,-38.065,431.916,171.049,28.924,155.430
C05041=1056.651,-38.314,431.929,171.047,28.922,155.429
C05042=1056.646,-38.564,431.942,171.046,28.920,155.429
C05043=1056.639,-38.814,431.955,171.044,28.918,155.429
C05044=1056.633,-39.064,431.968,171.042,28.917,155.429
C05045=1056.627,-39.313,431.981,171.040,28.915,155.429
C05046=1056.621,-39.563,431.994,171.039,28.913,155.428
C05047=1056.614,-39.812,432.007,171.037,28.911,155.428
C05048=1056.609,-40.062,432.019,171.035,28.909,155.428
C05049=1056.602,-40.311,432.032,171.033,28.908,155.428
C05050=1056.596,-40.561,432.045,171.032,28.906,155.428
C05051=1056.590,-40.811,432.057,171.030,28.904,155.428
C05052=1056.584,-41.060,432.071,171.028,28.902,155.427
C05053=1056.578,-41.310,432.083,171.026,28.900,155.427
C05054=1056.571,-41.559,432.096,171.025,28.899,155.427
C05055=1056.565,-41.809,432.108,171.023,28.897,155.427
C05056=1056.558,-42.058,432.122,171.021,28.895,155.427
C05057=1056.552,-42.308,432.134,171.019,28.893,155.426
C05058=1056.546,-42.558,432.147,171.018,28.892,155.426
C05059=1056.539,-42.807,432.160,171.016,28.889,155.426
C05060=1056.533,-43.057,432.172,171.014,28.888,155.426
C05061=1056.527,-43.306,432.186,171.012,28.886,155.426
C05062=1056.521,-43.556,432.198,171.011,28.884,155.425
C05063=1056.515,-43.806,432.211,171.009,28.882,155.425
C05064=1056.508,-44.055,432.223,171.007,28.881,155.425
C05065=1056.502,-44.305,432.236,171.005,28.879,155.425
C05066=1056.497,-44.555,432.248,171.004,28.877,155.425
C05067=1056.490,-44.804,432.262,171.002,28.875,155.425
C05068=1056.484,-45.054,432.274,171.000,28.874,155.424
C05069=1056.478,-45.304,432.286,170.998,28.872,155.424
C05070=1056.472,-45.553,432.299,170.997,28.870,155.424
C05071=1056.466,-45.803,432.312,170.995,28.868,155.424
C05072=1056.460,-46.053,432.325,170.993,28.867,155.424
C05073=1056.454,-46.301,432.336,170.991,28.865,155.424
C05074=1056.447,-46.551,432.349,170.990,28.863,155.423
C05075=1056.442,-46.801,432.362,170.988,28.861,155.423
C05076=1056.436,-47.050,432.375,170.986,28.859,155.423
C05077=1056.429,-47.300,432.387,170.984,28.858,155.423
C05078=1056.423,-47.549,432.400,170.983,28.856,155.423
C05079=1056.417,-47.799,432.412,170.981,28.854,155.422
C05080=1056.411,-48.049,432.425,170.979,28.852,155.422
C05081=1056.404,-48.299,432.437,170.977,28.851,155.422
C05082=1056.398,-48.548,432.450,170.976,28.849,155.422
C05083=1056.392,-48.798,432.463,170.974,28.847,155.422
C05084=1056.386,-49.048,432.475,170.972,28.845,155.422
C05085=1056.380,-49.297,432.487,170.970,28.844,155.421
C05086=1056.374,-49.546,432.499,170.969,28.842,155.421
C05087=1056.368,-49.796,432.513,170.967,28.840,155.421
C05088=1056.361,-50.045,432.525,170.965,28.838,155.421
C05089=1056.355,-50.326,432.539,170.963,28.836,155.421
C05090=1056.348,-50.605,432.552,170.962,28.835,155.421
C05091=1056.341,-50.886,432.567,170.959,28.832,155.420
C05092=1056.334,-51.165,432.580,170.957,28.831,155.420
C05093=1056.327,-51.414,432.592,170.955,28.829,155.420
C05094=1056.321,-51.664,432.605,170.954,28.827,155.420
C05095=1056.314,-51.914,432.617,170.952,28.826,155.420
C05096=1056.308,-52.164,432.629,170.950,28.824,155.420
C05097=1056.302,-52.413,432.641,170.948,28.823,155.419
C05098=1056.296,-52.663,432.654,170.947,28.821,155.419
C05099=1056.289,-52.913,432.666,170.945,28.819,155.419
C05100=1056.283,-53.162,432.678,170.943,28.818,155.419
C05101=1056.277,-53.412,432.690,170.941,28.817,155.419
C05102=1056.271,-53.661,432.702,170.939,28.815,155.419
C05103=1056.265,-53.911,432.715,170.938,28.813,155.419
C05104=1056.258,-54.161,432.726,170.936,28.812,155.418
C05105=1056.251,-54.410,432.738,170.934,28.810,155.418
C05106=1056.246,-54.660,432.751,170.932,28.809,155.418
C05107=1056.239,-54.910,432.763,170.931,28.807,155.418
C05108=1056.233,-55.159,432.776,170.929,28.805,155.418
C05109=1056.226,-55.409,432.787,170.926,28.803,155.418
C05110=1056.220,-55.658,432.799,170.924,28.802,155.418
C05111=1056.214,-55.908,432.812,170.923,28.800,155.417
C05112=1056.208,-56.157,432.824,170.921,28.798,155.417
C05113=1056.202,-56.407,432.836,170.919,28.797,155.417
C05114=1056.195,-56.657,432.848,170.917,28.795,155.417
C05115=1056.189,-56.906,432.860,170.916,28.794,155.417
C05116=1056.183,-57.156,432.873,170.914,28.793,155.417
C05117=1056.177,-57.406,432.883,170.912,28.791,155.417
C05118=1056.170,-57.655,432.895,170.910,28.789,155.417
C05119=1056.164,-57.905,432.908,170.908,28.788,155.416
C05120=1056.158,-58.155,432.920,170.907,28.786,155.416
C05121=1056.152,-58.405,432.932,170.905,28.784,155.416
C05122=1056.146,-58.654,432.944,170.903,28.783,155.416
C05123=1056.139,-58.903,432.956,170.901,28.781,155.416
C05124=1056.133,-59.153,432.969,170.900,28.780,155.416
C05125=1056.127,-59.403,432.980,170.898,28.778,155.416
C05126=1056.120,-59.653,432.992,170.896,28.777,155.415
C05127=1056.115,-59.902,433.004,170.894,28.775,155.415
C05128=1056.108,-60.151,433.016,170.892,28.774,155.415
C05129=1056.102,-60.401,433.028,170.891,28.772,155.415
C05130=1056.096,-60.651,433.040,170.889,28.770,155.415
C05131=1056.090,-60.900,433.051,170.887,28.769,155.415
C05132=1056.083,-61.150,433.063,170.884,28.767,155.415
C05133=1056.077,-61.400,433.076,170.883,28.766,155.415
C05134=1056.071,-61.649,433.088,170.881,28.764,155.414
C05135=1056.065,-61.899,433.099,170.879,28.762,155.414
C05136=1056.059,-62.149,433.111,170.877,28.761,155.414
C05137=1056.052,-62.398,433.123,170.876,28.760,155.414
C05138=1056.046,-62.648,433.135,170.874,28.758,155.414
C05139=1056.041,-62.898,433.147,170.872,28.757,155.414
C05140=1056.034,-63.147,433.159,170.870,28.755,155.414
C05141=1056.028,-63.397,433.171,170.868,28.753,155.414
C05142=1056.022,-63.646,433.183,170.867,28.752,155.413
C05143=1056.016,-63.896,433.194,170.865,28.751,155.413
C05144=1056.009,-64.146,433.206,170.863,28.749,155.413
C05145=1056.003,-64.395,433.218,170.861,28.747,155.413
C05146=1055.998,-64.645,433.229,170.860,28.746,155.413
C05147=1055.991,-64.895,433.241,170.858,28.745,155.413
C05148=1055.984,-65.144,433.253,170.856,28.743,155.413
C05149=1055.979,-65.394,433.265,170.854,28.741,155.413
C05150=1055.973,-65.644,433.277,170.852,28.740,155.412
C05151=1055.966,-65.893,433.289,170.850,28.739,155.412
C05152=1055.961,-66.143,433.300,170.848,28.737,155.412
C05153=1055.954,-66.424,433.313,170.846,28.735,155.412
C05154=1055.947,-66.705,433.327,170.844,28.734,155.412
C05155=1055.940,-66.986,433.340,170.842,28.732,155.412
C05156=1055.933,-67.267,433.353,170.840,28.730,155.412
C05157=1055.927,-67.517,433.364,170.838,28.728,155.412
C05158=1055.920,-67.767,433.376,170.836,28.727,155.411
C05159=1055.914,-68.016,433.388,170.835,28.726,155.411
C05160=1055.909,-68.266,433.400,170.833,28.724,155.411
C05161=1055.902,-68.516,433.412,170.831,28.723,155.411
C05162=1055.896,-68.765,433.423,170.829,28.721,155.411
C05163=1055.890,-69.015,433.435,170.827,28.720,155.411
C05164=1055.885,-69.265,433.446,170.826,28.718,155.411
C05165=1055.878,-69.514,433.458,170.824,28.717,155.411
C05166=1055.872,-69.764,433.469,170.821,28.715,155.411
C05167=1055.866,-70.013,433.481,170.819,28.714,155.410
C05168=1055.860,-70.264,433.493,170.818,28.712,155.410
C05169=1055.854,-70.513,433.504,170.816,28.711,155.410
C05170=1055.848,-70.763,433.515,170.814,28.709,155.410
C05171=1055.842,-71.012,433.527,170.812,28.708,155.410
C05172=1055.836,-71.262,433.539,170.810,28.707,155.410
C05173=1055.830,-71.511,433.550,170.809,28.705,155.410
C05174=1055.824,-71.761,433.562,170.807,28.703,155.410
C05175=1055.818,-72.010,433.573,170.805,28.702,155.410
C05176=1055.812,-72.261,433.585,170.803,28.701,155.409
C05177=1055.806,-72.511,433.596,170.802,28.699,155.409
C05178=1055.800,-72.760,433.608,170.800,28.698,155.409
C05179=1055.793,-73.010,433.619,170.798,28.696,155.409
C05180=1055.787,-73.259,433.631,170.796,28.695,155.409
C05181=1055.782,-73.509,433.643,170.793,28.693,155.409
C05182=1055.776,-73.758,433.654,170.792,28.692,155.409
C05183=1055.769,-74.008,433.665,170.790,28.691,155.409
C05184=1055.764,-74.258,433.676,170.788,28.689,155.409
C05185=1055.757,-74.508,433.688,170.786,28.688,155.409
C05186=1055.751,-74.757,433.699,170.784,28.686,155.408
C05187=1055.745,-75.007,433.710,170.783,28.685,155.408
C05188=1055.739,-75.256,433.722,170.781,28.684,155.408
C05189=1055.732,-75.506,433.733,170.779,28.683,155.408
C05190=1055.727,-75.756,433.744,170.777,28.681,155.408
C05191=1055.720,-76.005,433.756,170.775,28.680,155.408
C05192=1055.714,-76.256,433.767,170.774,28.678,155.408
C05193=1055.708,-76.505,433.778,170.771,28.677,155.408
C05194=1055.702,-76.755,433.789,170.769,28.676,155.408
C05195=1055.696,-77.004,433.801,170.767,28.675,155.408
C05196=1055.689,-77.254,433.812,170.765,28.673,155.408
C05197=1055.683,-77.504,433.823,170.764,28.672,155.408
C05198=1055.677,-77.754,433.834,170.762,28.671,155.408
C05199=1055.671,-78.003,433.846,170.760,28.669,155.407
C05200=1055.665,-78.253,433.857,170.758,28.668,155.407
C05201=1055.658,-78.502,433.868,170.756,28.667,155.407
C05202=1055.653,-78.752,433.878,170.755,28.665,155.407
C05203=1055.646,-79.001,433.890,170.753,28.664,155.407
C05204=1055.640,-79.251,433.901,170.750,28.663,155.407
C05205=1055.634,-79.501,433.913,170.748,28.661,155.407
C05206=1055.628,-79.750,433.923,170.746,28.660,155.407
C05207=1055.622,-80.001,433.935,170.745,28.659,155.407
C05208=1055.616,-80.250,433.946,170.743,28.658,155.407
C05209=1055.609,-80.499,433.957,170.741,28.657,155.407
C05210=1055.603,-80.749,433.968,170.739,28.656,155.407
C05211=1055.597,-80.999,433.979,170.737,28.654,155.407
C05212=1055.591,-81.249,433.990,170.736,28.653,155.407
C05213=1055.584,-81.498,434.001,170.734,28.652,155.407
C05214=1055.578,-81.748,434.011,170.731,28.651,155.407
C05215=1055.572,-81.998,434.023,170.729,28.650,155.407
C05216=1055.566,-82.248,434.034,170.727,28.648,155.406
C05217=1055.558,-82.531,434.046,170.726,28.647,155.406
C05218=1055.551,-82.814,434.059,170.723,28.646,155.406
C05219=1055.544,-83.098,434.071,170.721,28.644,155.406
C05220=1055.537,-83.381,434.083,170.719,28.643,155.406
C05221=1055.531,-83.630,434.094,170.717,28.642,155.406
C05222=1055.524,-83.880,434.104,170.715,28.641,155.406
C05223=1055.519,-84.130,434.115,170.713,28.640,155.406
C05224=1055.512,-84.380,434.127,170.711,28.638,155.406
C05225=1055.507,-84.630,434.137,170.709,28.637,155.406
C05226=1055.499,-84.879,434.149,170.707,28.636,155.406
C05227=1055.493,-85.128,434.160,170.705,28.635,155.406
C05228=1055.488,-85.378,434.170,170.704,28.634,155.406
C05229=1055.481,-85.628,434.180,170.702,28.633,155.406
C05230=1055.475,-85.878,434.191,170.700,28.632,155.406
C05231=1055.469,-86.128,434.203,170.698,28.630,155.406
C05232=1055.462,-86.377,434.213,170.695,28.629,155.406
C05233=1055.457,-86.627,434.224,170.694,28.628,155.406
C05234=1055.450,-86.877,434.235,170.692,28.627,155.406
C05235=1055.444,-87.126,434.245,170.690,28.626,155.406
C05236=1055.438,-87.375,434.256,170.688,28.625,155.406
C05237=1055.432,-87.626,434.267,170.686,28.624,155.405
C05238=1055.425,-87.875,434.278,170.684,28.623,155.405
C05239=1055.419,-88.125,434.289,170.683,28.622,155.405
C05240=1055.413,-88.375,434.300,170.680,28.620,155.405
C05241=1055.407,-88.624,434.310,170.678,28.619,155.405
C05242=1055.400,-88.874,434.321,170.676,28.618,155.405
C05243=1055.395,-89.124,434.332,170.674,28.617,155.405
C05244=1055.388,-89.373,434.342,170.673,28.616,155.405
C05245=1055.383,-89.623,434.353,170.671,28.614,155.405
C05246=1055.376,-89.873,434.364,170.669,28.613,155.405
C05247=1055.370,-90.122,434.374,170.667,28.612,155.405
C05248=1055.364,-90.372,434.385,170.665,28.611,155.405
C05249=1055.358,-90.622,434.396,170.662,28.610,155.405
C05250=1055.352,-90.872,434.406,170.661,28.609,155.405
C05251=1055.346,-91.121,434.417,170.659,28.608,155.405
C05252=1055.339,-91.371,434.427,170.657,28.607,155.405
C05253=1055.333,-91.620,434.438,170.655,28.606,155.405
C05254=1055.327,-91.870,434.449,170.653,28.605,155.405
C05255=1055.321,-92.120,434.459,170.651,28.604,155.405
C05256=1055.315,-92.370,434.470,170.650,28.603,155.405
C05257=1055.309,-92.619,434.481,170.648,28.602,155.405
C05258=1055.303,-92.869,434.491,170.645,28.600,155.405
C05259=1055.297,-93.119,434.501,170.643,28.599,155.405
C05260=1055.290,-93.369,434.512,170.641,28.598,155.405
C05261=1055.284,-93.618,434.523,170.639,28.597,155.405
C05262=1055.279,-93.867,434.534,170.638,28.596,155.405
C05263=1055.272,-94.117,434.543,170.636,28.595,155.405
C05264=1055.266,-94.367,434.555,170.634,28.594,155.405
C05265=1055.260,-94.617,434.565,170.632,28.593,155.405
C05266=1055.254,-94.867,434.575,170.629,28.592,155.405
C05267=1055.248,-95.116,434.586,170.627,28.591,155.405
C05268=1055.242,-95.365,434.596,170.626,28.590,155.405
C05269=1055.236,-95.616,434.607,170.624,28.589,155.405
C05270=1055.229,-95.865,434.617,170.622,28.588,155.404
C05271=1055.224,-96.115,434.628,170.620,28.587,155.404
C05272=1055.218,-96.365,434.638,170.618,28.586,155.404
C05273=1055.212,-96.614,434.648,170.616,28.585,155.404
C05274=1055.206,-96.864,434.659,170.615,28.584,155.404
C05275=1055.199,-97.114,434.669,170.612,28.583,155.404
C05276=1055.194,-97.364,434.680,170.610,28.582,155.404
C05277=1055.187,-97.613,434.690,170.608,28.581,155.404
C05278=1055.182,-97.863,434.700,170.606,28.580,155.404
C05279=1055.175,-98.112,434.711,170.604,28.579,155.404
C05280=1055.168,-98.363,434.721,170.603,28.578,155.404
C05281=1055.162,-98.647,434.733,170.600,28.577,155.404
C05282=1055.155,-98.933,434.744,170.598,28.576,155.404
C05283=1055.148,-99.219,434.756,170.595,28.575,155.404
C05284=1055.140,-99.505,434.768,170.593,28.574,155.404
C05285=1055.134,-99.754,434.778,170.591,28.573,155.404
C05286=1055.128,-100.004,434.788,170.590,28.572,155.404
C05287=1055.122,-100.254,434.798,170.588,28.571,155.404
C05288=1055.115,-100.504,434.809,170.585,28.570,155.405
C05289=1055.110,-100.754,434.819,170.583,28.569,155.405
C05290=1055.103,-101.003,434.829,170.581,28.568,155.404
C05291=1055.098,-101.253,434.839,170.579,28.567,155.404
C05292=1055.091,-101.502,434.850,170.577,28.567,155.405
C05293=1055.085,-101.752,434.859,170.576,28.566,155.405
C05294=1055.079,-102.001,434.870,170.574,28.565,155.404
C05295=1055.073,-102.252,434.880,170.572,28.564,155.405
C05296=1055.066,-102.502,434.889,170.569,28.563,155.405
C05297=1055.060,-102.751,434.900,170.567,28.562,155.405
C05298=1055.055,-103.001,434.910,170.565,28.562,155.405
C05299=1055.048,-103.250,434.920,170.564,28.561,155.405
C05300=1055.042,-103.500,434.930,170.562,28.560,155.405
C05301=1055.036,-103.749,434.941,170.560,28.559,155.405
C05302=1055.030,-103.999,434.950,170.558,28.558,155.405
C05303=1055.023,-104.250,434.960,170.555,28.557,155.405
C05304=1055.017,-104.499,434.971,170.553,28.556,155.405
C05305=1055.011,-104.749,434.981,170.551,28.555,155.405
C05306=1055.005,-104.999,434.990,170.550,28.555,155.405
C05307=1054.999,-105.248,435.000,170.548,28.554,155.405
C05308=1054.993,-105.498,435.011,170.546,28.553,155.405
C05309=1054.987,-105.748,435.020,170.544,28.552,155.405
C05310=1054.981,-105.997,435.030,170.541,28.552,155.405
C05311=1054.974,-106.247,435.040,170.539,28.551,155.405
C05312=1054.969,-106.497,435.050,170.537,28.550,155.405
C05313=1054.962,-106.746,435.060,170.536,28.549,155.405
C05314=1054.956,-106.996,435.070,170.534,28.548,155.405
C05315=1054.950,-107.246,435.080,170.532,28.548,155.405
C05316=1054.944,-107.495,435.090,170.530,28.547,155.405
C05317=1054.938,-107.745,435.100,170.528,28.546,155.405
C05318=1054.931,-107.996,435.110,170.525,28.545,155.405
C05319=1054.925,-108.245,435.120,170.523,28.544,155.405
C05320=1054.919,-108.495,435.130,170.521,28.544,155.405
C05321=1054.913,-108.744,435.139,170.520,28.543,155.405
C05322=1054.906,-108.994,435.149,170.518,28.542,155.405
C05323=1054.901,-109.244,435.159,170.516,28.541,155.405
C05324=1054.895,-109.493,435.169,170.513,28.541,155.405
C05325=1054.888,-109.743,435.179,170.511,28.540,155.405
C05326=1054.882,-109.993,435.189,170.509,28.539,155.405
C05327=1054.876,-110.243,435.198,170.507,28.539,155.406
C05328=1054.870,-110.493,435.208,170.506,28.538,155.405
C05329=1054.864,-110.742,435.217,170.504,28.537,155.406
C05330=1054.857,-110.992,435.228,170.502,28.537,155.406
C05331=1054.851,-111.241,435.237,170.499,28.536,155.406
C05332=1054.846,-111.492,435.247,170.497,28.535,155.406
C05333=1054.839,-111.741,435.257,170.495,28.535,155.406
C05334=1054.833,-111.991,435.266,170.493,28.534,155.406
C05335=1054.827,-112.241,435.276,170.491,28.533,155.406
C05336=1054.821,-112.491,435.286,170.490,28.532,155.406
C05337=1054.814,-112.740,435.296,170.488,28.532,155.406
C05338=1054.808,-112.990,435.305,170.485,28.531,155.406
C05339=1054.802,-113.240,435.315,170.483,28.530,155.406
C05340=1054.796,-113.489,435.325,170.481,28.530,155.406
C05341=1054.790,-113.739,435.334,170.479,28.529,155.406
C05342=1054.784,-113.989,435.344,170.477,28.529,155.406
C05343=1054.777,-114.239,435.353,170.475,28.528,155.406
C05344=1054.771,-114.489,435.363,170.473,28.527,155.406
C05345=1054.764,-114.772,435.374,170.471,28.527,155.406
C05346=1054.758,-115.056,435.384,170.469,28.526,155.406
C05347=1054.750,-115.341,435.395,170.466,28.525,155.407
C05348=1054.743,-115.624,435.406,170.464,28.524,155.407
C05349=1054.737,-115.874,435.416,170.462,28.524,155.407
C05350=1054.731,-116.124,435.425,170.459,28.523,155.407
C05351=1054.725,-116.374,435.435,170.457,28.522,155.407
C05352=1054.719,-116.624,435.445,170.455,28.522,155.407
C05353=1054.713,-116.873,435.454,170.454,28.521,155.407
C05354=1054.706,-117.123,435.464,170.452,28.521,155.407
C05355=1054.700,-117.373,435.473,170.450,28.521,155.407
C05356=1054.694,-117.623,435.483,170.448,28.520,155.407
C05357=1054.689,-117.872,435.491,170.445,28.519,155.407
C05358=1054.683,-118.122,435.501,170.443,28.518,155.407
C05359=1054.677,-118.372,435.510,170.441,28.518,155.407
C05360=1054.670,-118.622,435.520,170.439,28.518,155.408
C05361=1054.664,-118.872,435.530,170.437,28.517,155.408
C05362=1054.658,-119.121,435.539,170.436,28.517,155.408
C05363=1054.652,-119.371,435.549,170.433,28.516,155.408
C05364=1054.645,-119.621,435.558,170.431,28.515,155.408
C05365=1054.639,-119.870,435.567,170.429,28.515,155.408
C05366=1054.633,-120.120,435.576,170.427,28.514,155.408
C05367=1054.627,-120.369,435.586,170.425,28.514,155.408
C05368=1054.621,-120.620,435.595,170.423,28.513,155.408
C05369=1054.615,-120.870,435.604,170.421,28.513,155.408
C05370=1054.609,-121.119,435.614,170.418,28.512,155.408
C05371=1054.603,-121.369,435.624,170.417,28.512,155.408
C05372=1054.596,-121.619,435.633,170.415,28.511,155.409
C05373=1054.590,-121.868,435.642,170.413,28.511,155.409
C05374=1054.584,-122.118,435.651,170.411,28.510,155.409
C05375=1054.578,-122.368,435.660,170.409,28.510,155.409
C05376=1054.572,-122.618,435.670,170.406,28.509,155.409
C05377=1054.566,-122.868,435.679,170.404,28.509,155.409
C05378=1054.560,-123.117,435.689,170.402,28.508,155.409
C05379=1054.554,-123.367,435.697,170.400,28.508,155.409
C05380=1054.547,-123.617,435.706,170.398,28.507,155.409
C05381=1054.541,-123.866,435.716,170.396,28.507,155.409
C05382=1054.535,-124.116,435.725,170.395,28.507,155.409
C05383=1054.529,-124.367,435.734,170.392,28.506,155.410
C05384=1054.523,-124.615,435.743,170.390,28.505,155.410
C05385=1054.517,-124.865,435.753,170.388,28.505,155.410
C05386=1054.511,-125.116,435.761,170.386,28.505,155.410
C05387=1054.505,-125.365,435.771,170.384,28.504,155.410
C05388=1054.498,-125.615,435.780,170.382,28.504,155.410
C05389=1054.492,-125.864,435.789,170.379,28.504,155.410
C05390=1054.486,-126.114,435.798,170.377,28.503,155.410
C05391=1054.479,-126.364,435.807,170.375,28.503,155.410
C05392=1054.473,-126.614,435.817,170.373,28.502,155.410
C05393=1054.468,-126.863,435.825,170.372,28.502,155.411
C05394=1054.462,-127.113,435.835,170.370,28.501,155.411
C05395=1054.455,-127.363,435.844,170.367,28.501,155.411
C05396=1054.449,-127.613,435.852,170.365,28.501,155.411
C05397=1054.443,-127.863,435.862,170.363,28.501,155.411
C05398=1054.438,-128.113,435.871,170.361,28.499,155.411
C05399=1054.434,-128.363,435.881,170.359,28.498,155.411
C05400=1054.432,-128.612,435.893,170.358,28.496,155.411
C05401=1054.430,-128.863,435.905,170.356,28.493,155.410
C05402=1054.430,-129.114,435.916,170.355,28.491,155.410
C05403=1054.432,-129.364,435.930,170.354,28.487,155.409
C05404=1054.433,-129.614,435.944,170.352,28.483,155.409
C05405=1054.437,-129.865,435.958,170.352,28.479,155.408
C05406=1054.441,-130.117,435.973,170.351,28.473,155.407
C05407=1054.447,-130.368,435.989,170.351,28.467,155.406
C05408=1054.454,-130.617,436.005,170.350,28.461,155.405
C05409=1054.083,-130.640,435.793,170.303,28.629,155.438
C05410=1054.076,-130.390,435.776,170.303,28.635,155.439
C05411=1054.070,-130.140,435.761,170.304,28.640,155.440
C05412=1054.066,-129.889,435.746,170.305,28.646,155.441
C05413=1054.062,-129.637,435.731,170.305,28.650,155.442
C05414=1054.061,-129.387,435.718,170.307,28.654,155.442
C05415=1054.059,-129.137,435.705,170.307,28.658,155.443
C05416=1054.060,-128.887,435.692,170.309,28.661,155.443
C05417=1054.061,-128.635,435.681,170.310,28.663,155.444
C05418=1054.063,-128.386,435.669,170.312,28.666,155.444
C05419=1054.067,-128.136,435.658,170.314,28.667,155.444
C05420=1054.072,-127.886,435.648,170.316,28.668,155.444
C05421=1054.077,-127.636,435.640,170.318,28.668,155.444
C05422=1054.084,-127.386,435.631,170.320,28.669,155.444
C05423=1054.090,-127.137,435.621,170.322,28.669,155.444
C05424=1054.096,-126.886,435.612,170.325,28.669,155.444
C05425=1054.103,-126.637,435.604,170.326,28.669,155.443
C05426=1054.109,-126.388,435.594,170.328,28.670,155.443
C05427=1054.115,-126.137,435.585,170.330,28.670,155.443
C05428=1054.121,-125.887,435.576,170.332,28.671,155.443
C05429=1054.127,-125.639,435.567,170.334,28.671,155.443
C05430=1054.133,-125.388,435.558,170.337,28.672,155.443
C05431=1054.139,-125.138,435.549,170.339,28.672,155.443
C05432=1054.146,-124.889,435.540,170.341,28.672,155.443
C05433=1054.152,-124.639,435.531,170.343,28.672,155.443
C05434=1054.157,-124.389,435.522,170.345,28.673,155.443
C05435=1054.164,-124.140,435.512,170.347,28.673,155.442
C05436=1054.170,-123.890,435.503,170.348,28.674,155.442
C05437=1054.176,-123.640,435.494,170.351,28.674,155.442
C05438=1054.183,-123.390,435.485,170.353,28.675,155.442
C05439=1054.188,-123.141,435.476,170.355,28.675,155.442
C05440=1054.194,-122.891,435.466,170.357,28.676,155.442
C05441=1054.201,-122.641,435.457,170.359,28.676,155.442
C05442=1054.206,-122.391,435.448,170.361,28.677,155.442
C05443=1054.213,-122.141,435.439,170.364,28.677,155.442
C05444=1054.219,-121.892,435.429,170.366,28.678,155.442
C05445=1054.225,-121.642,435.420,170.368,28.678,155.442
C05446=1054.231,-121.393,435.410,170.370,28.678,155.441
C05447=1054.237,-121.142,435.402,170.371,28.679,155.441
C05448=1054.243,-120.892,435.392,170.373,28.679,155.441
C05449=1054.249,-120.643,435.382,170.376,28.680,155.441
C05450=1054.256,-120.393,435.373,170.378,28.680,155.441
C05451=1054.263,-120.143,435.364,170.380,28.681,155.441
C05452=1054.268,-119.894,435.355,170.382,28.681,155.441
C05453=1054.274,-119.644,435.345,170.384,28.682,155.441
C05454=1054.280,-119.394,435.336,170.386,28.683,155.441
C05455=1054.286,-119.144,435.327,170.389,28.683,155.441
C05456=1054.292,-118.894,435.317,170.390,28.684,155.441
C05457=1054.299,-118.645,435.308,170.392,28.684,155.441
C05458=1054.305,-118.395,435.298,170.394,28.685,155.441
C05459=1054.311,-118.145,435.288,170.396,28.685,155.440
C05460=1054.317,-117.896,435.280,170.398,28.686,155.440
